// TIA Portal project "GME" (V18)

(* hardware
DEVICE "S7-1500/ET200MP station_1"  S7-1500 station
   slot 0: "Rail_0"  Rack  6ES7 590-1***0-0AA0
   slot 1: "102CPU"  CPU 1515-2 PN  6ES7 515-2AN03-0AB0  V3.0
      slot 3: "CPU display_1"  6ES7591-1BA00-0AA0
      slot 32768: "PROFINET interface_1"  X1
         slot 32769: "Port_1"  X1 P1
         slot 32770: "Port_2"  X1 P2
      slot 33024: "PROFINET interface_2"  X2
         slot 33025: "Port_1"  X2 P1
      slot 34817: "Virtual CP interface port_1"  Virtual CP interface port  Virtual CP interface port
   slot 2: "102A1"  AI 8xU/I/RTD/TC ST  6ES7 531-7KF00-0AB0  V2.2
   slot 3: "102A2"  AI 8xU/I/RTD/TC ST  6ES7 531-7KF00-0AB0  V2.2
   slot 4: "102A3"  AI 8xU/I/RTD/TC ST  6ES7 531-7KF00-0AB0  V2.2
   slot 5: "102A4"  AI 8xU/I/RTD/TC ST  6ES7 531-7KF00-0AB0  V2.2
   slot 6: "102A5"  AQ 8xU/I HS  6ES7 532-5HF00-0AB0  V2.2
   slot 7: "102A6"  AQ 8xU/I HS  6ES7 532-5HF00-0AB0  V2.2
   slot 8: "102A7"  DI 32x24VDC HF  6ES7 521-1BL00-0AB0  V2.2
   slot 9: "102A8"  DI 32x24VDC HF  6ES7 521-1BL00-0AB0  V2.2
   slot 10: "103A1"  DI 32x24VDC HF  6ES7 521-1BL00-0AB0  V2.2
   slot 11: "103A2"  DI 32x24VDC HF  6ES7 521-1BL00-0AB0  V2.2
   slot 12: "103A3"  DI 32x24VDC HF  6ES7 521-1BL00-0AB0  V2.2
   slot 13: "103GD1"  PS 25W 24VDC  6ES7 505-0KA00-0AB0  V1.0
   slot 14: "103A4"  DQ 32x24VDC/0.5A HF  6ES7 522-1BL01-0AB0  V1.1
   slot 15: "103A5"  DQ 32x24VDC/0.5A HF  6ES7 522-1BL01-0AB0  V1.1
   slot 16: "103A6"  TM Count 2x24V  6ES7 550-1AA01-0AB0  V2.0
   slot 17: "103A7"  TM Count 2x24V  6ES7 550-1AA01-0AB0  V2.0
   slot 18: "103A8"  TM Count 2x24V  6ES7 550-1AA01-0AB0  V2.0
DEVICE "S7-1500/ET200MP station_2"  S7-1500 station
   slot 0: "Rail_0"  Rack  6ES7 590-1***0-0AA0
   slot 1: "153IM155_JB1"  IM 155-5 PN ST  6ES7 155-5AA01-0AB0  V4.1
   slot 2: "153A1"  AI 8xU/I/RTD/TC ST  6ES7 531-7KF00-0AB0  V2.2
   slot 3: "153A2"  DQ 32x24VDC/0.5A HF  6ES7 522-1BL01-0AB0  V1.1
   slot 4: "153A3"  DI 16x24VDC/DQ 16x24VDC/0.5A BA  6ES7 523-1BL00-0AA0  V1.1
   slot 5: "153A4"  AQ 8xU/I HS  6ES7 532-5HF00-0AB0  V2.2
DEVICE "S7-1500/ET200MP station_3"  S7-1500 station
   slot 0: "Rail_0"  Rack  6ES7 590-1***0-0AA0
   slot 1: "182IM155_JB2"  IM 155-5 PN ST  6ES7 155-5AA01-0AB0  V4.1
   slot 2: "182A1"  DQ 32x24VDC/0.5A HF  6ES7 522-1BL01-0AB0  V1.1
   slot 3: "182A2"  DI 16x24VDC/DQ 16x24VDC/0.5A BA  6ES7 523-1BL00-0AA0  V1.1
*)

// ===== PLC "102CPU"  CPU 1515-2 PN =====

VAR_GLOBAL   // PLC tag table "Default tag table"
   "Main flame ON" AT %M25.0 : Bool;
   "Flag AutoBurner" AT %M15.0 : Bool;
   "Flag_Aggiorna_DB" AT %M1.7 : Bool;
   "Stop Counter PEW 336" AT %M114.3 : Bool;
   "Stop Counter PEW 368" AT %M115.3 : Bool;
   "Stop Counter PEW 418" AT %M116.3 : Bool;
   "TC01-TC02control disable" AT %M80.2 : Bool;
   "TC03 Close" AT %M40.7 : Bool;
   "TC03 Close2" AT %M41.1 : Bool;
   "TC03 Open" AT %M40.6 : Bool;
   "TC03 Open2" AT %M41.0 : Bool;
   "TEST CABIN" AT %M5.0 : Bool;
   "EV-82" AT %Q21.7 : Bool;   // A11.7 FILTER 8 VALVE BF02FOURTH SECTOR
   "EV-83" AT %Q22.0 : Bool;   // A12.0 FILTER 1 VALVE BF02FIFTH SECTOR
   "EV-84" AT %Q22.1 : Bool;   // A12.1 FILTER 2 VALVE BF02FIFTH SECTOR
   "EV-85" AT %Q22.2 : Bool;   // A12.2 FILTER 3 VALVE BF02FIFTH SECTOR
   "EV-87" AT %Q22.4 : Bool;   // A12.4 FILTER 5 VALVE BF02FIFTH SECTOR
   "EV-88" AT %Q22.5 : Bool;   // A12.5 FILTER 6 VALVE BF02FIFTH SECTOR
   "EV-89" AT %Q22.6 : Bool;   // A12.6 FILTER 7 VALVE BF02FIFTH SECTOR
   "EV-90" AT %Q22.7 : Bool;   // A12.7 FILTER 8 VALVE BF02FIFTH SECTOR
   "Module Access FLT" AT %M32.3 : Bool;
   "OB Fault" AT %M32.1 : Bool;
   "OFF" AT %M0.1 : Bool;
   "ON" AT %M0.0 : Bool;
   "OPEN MV05 PID" AT %M11.4 : Bool;
   "Every 1 second" AT %M1.0 : Bool;
   "Open EV A 00 PV-01" AT %M20.0 : Bool;
   "Open EV A 00 PV-02" AT %M30.4 : Bool;
   "Open EV A 01  PV-01" AT %M21.3 : Bool;
   "Riduce MN01" AT %M1.2 : Bool;
   "Scarico ceneri auto" AT %M15.1 : Bool;
   "Braking VS01" AT %Q49.5 : Bool;   // It's no longer there
   "Start Burner" AT %M48.3 : Bool;
   "PID DOWN MV04" AT %M14.3 : Bool;
   "PID DOWN MV05" AT %M13.1 : Bool;
   "PID MV02 Down" AT %M14.1 : Bool;
   "PID MV02 UP" AT %M14.0 : Bool;
   "PID UP MV03" AT %M14.4 : Bool;
   "PID UP MV04" AT %M14.2 : Bool;
   "PID UP MV05" AT %M13.0 : Bool;
   "PID down MV03" AT %M14.5 : Bool;
   "MEM2_0" AT %M2.0 : Bool;
   "MV WORK PULSE" AT %M10.0 : Bool;
   "WASHING MAX OK" AT %M9.0 : Bool;
   "PV-02 Gate ON" AT %M12.2 : Bool;
   "Close EV A 00  PV-01" AT %M20.2 : Bool;
   "Close EV A 01  PV-01" AT %M21.0 : Bool;
   "Close EV A 01  PV-02" AT %M30.0 : Bool;
   "Close EV A 02  PV-01" AT %M22.3 : Bool;
   "Close EV B 00  PV-01" AT %M20.3 : Bool;
   "Close EV B 01  PV-01" AT %M21.2 : Bool;
   "Close EV B 01  PV-02" AT %M30.2 : Bool;
   "Close EV B 02  PV-01" AT %M22.1 : Bool;
   "Close MV02 PID" AT %M11.7 : Bool;
   "Enable Counter PEW 336" AT %M114.2 : Bool;
   "Enable Counter PEW 368" AT %M115.2 : Bool;
   "Enable Counter PEW 418" AT %M116.2 : Bool;
   "Start VS01 BRAKE" AT %M11.0 : Bool;
   "Start client motor 4" AT %Q61.2 : Bool;   // It should be Free but it is used
   "Start client motor 6" AT %Q61.3 : Bool;   // It should be Free but it is used
   "Start client motor 8" AT %Q61.4 : Bool;   // It should be Free but it is used
   "Start client motor 9" AT %Q61.5 : Bool;   // It should be Free but it is used
   "Start client motore 10" AT %Q61.6 : Bool;   // It should be Free but it is used
   "EV-66" AT %Q19.7 : Bool;   // A9.7 FILTER 8 VALVE BF02SECOND SECTOR
   "EV-67" AT %Q20.0 : Bool;   // A10.0 FILTER 1 VALVE BF02THIRD SECTOR
   "EV-68" AT %Q20.1 : Bool;   // A10.1 FILTER 2 VALVE BF02THIRD SECTOR
   "EV-69" AT %Q20.2 : Bool;   // A10.2 FILTER 3 VALVE BF02THIRD SECTOR
   "EV-70" AT %Q20.3 : Bool;   // A10.3 FILTER 4 VALVE BF02THIRD SECTOR
   "EV-71" AT %Q20.4 : Bool;   // A10.4 FILTER 5 VALVE BF02THIRD SECTOR
   "EV-72" AT %Q20.5 : Bool;   // A10.5 FILTER 6 VALVE BF02THIRD SECTOR
   "EV-73" AT %Q20.6 : Bool;   // A10.6 FILTER 7 VALVE BF02THIRD SECTOR
   "EV-74" AT %Q20.7 : Bool;   // A10.7 FILTER 8 VALVE BF02THIRD SECTOR
   "EV-75" AT %Q21.0 : Bool;   // A11.0 FILTER 1 VALVE BF02FOURTH SECTOR
   "Open EV B 00  PV-02" AT %M30.5 : Bool;
   "Open EV B 01  PV-01" AT %M21.1 : Bool;
   "Open EV B 01  PV-02" AT %M30.1 : Bool;
   "Open EV B 02  PV-01" AT %M22.2 : Bool;
   "Open MV02 PID" AT %M11.6 : Bool;
   "PC01 Close" AT %M40.2 : Bool;
   "PC01 Open" AT %M40.3 : Bool;
   "PC02 Close" AT %M40.4 : Bool;
   "PC02 Open" AT %M40.5 : Bool;
   "m491" AT %M10.1 : Bool;
   "maintenance PV01" AT %M80.5 : Bool;
   "maintenance PV02" AT %M80.6 : Bool;
   "PLS M51 6" AT %M51.6 : Bool;
   "PLS M51.5" AT %M51.5 : Bool;
   "PLS M51_4" AT %M51.4 : Bool;
   "PLS m10.3" AT %M10.3 : Bool;
   "PLS m10.4" AT %M10.4 : Bool;
   "Button pushed" AT %M60.0 : Bool;
   "CLOSE MV05 PID" AT %M11.5 : Bool;
   "PLS 50 3" AT %M50.3 : Bool;
   "PLS 50 4" AT %M50.4 : Bool;
   "PLS 50 6" AT %M50.6 : Bool;
   "PLS 50 7" AT %M50.7 : Bool;
   "PLS 50_5" AT %M50.5 : Bool;
   "PLS 51 1" AT %M51.1 : Bool;
   "PLS 51 2" AT %M51.2 : Bool;
   "PLS 51 3" AT %M51.3 : Bool;
   "PLS M50.0" AT %M50.0 : Bool;
   "PLS M50.1" AT %M50.1 : Bool;
   "PLS M50.2" AT %M50.2 : Bool;
   "PLS M51 0" AT %M51.0 : Bool;
   "EV-76" AT %Q21.1 : Bool;   // A11.1 FILTER 2 VALVE BF02FOURTH SECTOR
   "EV-77" AT %Q21.2 : Bool;   // A11.2 FILTER 3 VALVE BF02FOURTH SECTOR
   "EV-78" AT %Q21.3 : Bool;   // A11.3 FILTER 4 VALVE BF02FOURTH SECTOR
   "EV-79" AT %Q21.4 : Bool;   // A11.4 FILTER 5 VALVE BF02FOURTH SECTOR
   "EV-80" AT %Q21.5 : Bool;   // A11.5 FILTER 6 VALVE BF02FOURTH SECTOR
   "EV-81" AT %Q21.6 : Bool;   // A11.6 FILTER 7 VALVE BF02FOURTH SECTOR
   "EV-51" AT %Q18.0 : Bool;   // A8.0 FILTER 1 VALVE BF02FIRST SECTOR
   "EV-52" AT %Q18.1 : Bool;   // A8.1 FILTER 2 VALVE BF02FIRST SECTOR
   "EV-53" AT %Q18.2 : Bool;   // A8.2 FILTER 3 VALVE BF02FIRST SECTOR
   "EV-54" AT %Q18.3 : Bool;   // A8.3 FILTER 4 VALVE BF02FIRST SECTOR
   "EV-55" AT %Q18.4 : Bool;   // A8.4 FILTER 5 VALVE BF02FIRST SECTOR
   "EV-56" AT %Q18.5 : Bool;   // A8.5 FILTER 6 VALVE BF02FIRST SECTOR
   "EV-57" AT %Q18.6 : Bool;   // A8.6 FILTER 7 VALVE BF02FIRST SECTOR
   "EV-58" AT %Q18.7 : Bool;   // A8.7 FILTER 8 VALVE BF02FIRST SECTOR
   "EV-59" AT %Q19.0 : Bool;   // A9.0 FILTER 1 VALVE BF02SECOND SECTOR
   "MV06 PID DOWN" AT %M13.3 : Bool;
   "MV06 PID UP" AT %M13.2 : Bool;
   "MEM Gate A OPEN PV-01" AT %M10.7 : Bool;
   "MEM Gate A OPEN PV-02" AT %M12.4 : Bool;
   "MEM Gate B OPEN PV-01" AT %M10.6 : Bool;
   "MEM Gate B OPEN PV-02" AT %M12.3 : Bool;
   "RO01 Close" AT %M40.1 : Bool;
   "RO01 Open" AT %M40.0 : Bool;
   "RO01-RO02control disable" AT %M80.1 : Bool;
   "RO01_CLOSE" AT %M41.3 : Bool;
   "RO01_OPEN" AT %M41.2 : Bool;
   "Rack FAULT" AT %M32.2 : Bool;
   "Reset Counter PEW 336" AT %M114.5 : Bool;
   "Reset Counter PEW 368" AT %M115.5 : Bool;
   "Reset Counter PEW 418" AT %M116.5 : Bool;
   "Disable masses" AT %M80.0 : Bool;
   "EV-61" AT %Q19.2 : Bool;   // A9.2 FILTER 3 VALVE BF02SECOND SECTOR
   "EV-86" AT %Q22.3 : Bool;   // A12.3 FILTER 4 VALVE BF02FIFTH SECTOR
   "I/O FLT" AT %M32.0 : Bool;
   "UNDER TESTING" AT %M5.5 : Bool;
   "Init_RK_512" AT %M200.0 : Bool;
   "UP MV01 PID" AT %M12.0 : Bool;
   "UP MV04 PID" AT %M11.2 : Bool;
   "APP M10.2" AT %M10.2 : Bool;
   "Enable start burner" AT %M48.2 : Bool;
   "Open MV03 for washing" AT %M48.1 : Bool;
   "Open false air" AT %M2.1 : Bool;
   "Programmed stop burner" AT %M1.1 : Bool;
   "Open EV A 01  PV-02" AT %M30.3 : Bool;
   "Open EV A 02  PV-01" AT %M22.0 : Bool;
   "Open EV B 00  PV-01" AT %M20.1 : Bool;
   "Enable start burner(1)" AT %M48.0 : Bool;
   "Prog FAULT" AT %M32.4 : Bool;
   "R1 Gate ON" AT %M10.5 : Bool;
   "Shot to close" AT %M18.0 : Bool;
   "Shot to open" AT %M18.1 : Bool;
   "Counter error PEW 336" AT %M114.4 : Bool;
   "Counter error PEW 368" AT %M115.4 : Bool;
   "Counter error PEW 418" AT %M116.4 : Bool;
   "DOWN MV01 PID" AT %M12.1 : Bool;
   "DOWN MV04 PID" AT %M11.3 : Bool;
   "DOWN TC03 PID MV04" AT %M11.1 : Bool;
   "Lock Burner" AT %M28.0 : Bool;
   "EV-60" AT %Q19.1 : Bool;   // A9.1 FILTER 2 VALVE BF02SECOND SECTOR
   "EV-62" AT %Q19.3 : Bool;   // A9.3 FILTER 4 VALVE BF02SECOND SECTOR
   "EV-63" AT %Q19.4 : Bool;   // A9.4 FILTER 5 VALVE BF02SECOND SECTOR
   "EV-64" AT %Q19.5 : Bool;   // A9.5 FILTER 6 VALVE BF02SECOND SECTOR
   "EV-65" AT %Q19.6 : Bool;   // A9.6 FILTER 7 VALVE BF02SECOND SECTOR
   "Tag_47" AT %T13 : Timer;
   "Tag_48" AT %T17 : Timer;
   "Tag_49" AT %T120 : Timer;
   "Tag_50" AT %T121 : Timer;
   "Tag_51" AT %T39 : Timer;
   "Tag_52" AT %T99 : Timer;
   "Tag_53" AT %T101 : Timer;
   "Tag_54" AT %T49 : Timer;
   "Tag_55" AT %T52 : Timer;
   "Tag_56" AT %T53 : Timer;
   "Tag_57" AT %T54 : Timer;
   "Tag_58" AT %T55 : Timer;
   "Tag_59" AT %T60 : Timer;
   "Tag_60" AT %T61 : Timer;
   "Tag_61" AT %T62 : Timer;
   "Tag_62" AT %T63 : Timer;
   "Tag_63" AT %T66 : Timer;
   "Tag_64" AT %T67 : Timer;
   "Tag_65" AT %T70 : Timer;
   "Tag_66" AT %T71 : Timer;
   "Tag_67" AT %T91 : Timer;
   "Tag_68" AT %T72 : Timer;
   "Tag_69" AT %T73 : Timer;
   "Tag_70" AT %T75 : Timer;
   "Tag_71" AT %T80 : Timer;
   "Tag_72" AT %T81 : Timer;
   "Tag_73" AT %T82 : Timer;
   "Tag_74" AT %T83 : Timer;
   "Tag_75" AT %T84 : Timer;
   "Tag_76" AT %T93 : Timer;
   "Tag_77" AT %T94 : Timer;
   "Tag_78" AT %T95 : Timer;
   "Tag_79" AT %T96 : Timer;
   "Tag_80" AT %T103 : Timer;
   "Tag_81" AT %T104 : Timer;
   "Tag_82" AT %T105 : Timer;
   "Tag_83" AT %T106 : Timer;
   "Tag_84" AT %T107 : Timer;
   "Tag_85" AT %T108 : Timer;
   "Tag_86" AT %T109 : Timer;
   "Tag_87" AT %T110 : Timer;
   "Tag_88" AT %T111 : Timer;
   "Tag_89" AT %T112 : Timer;
   "Tag_90" AT %T43 : Timer;
   "Tag_91" AT %T44 : Timer;
   "Tag_92" AT %T4 : Timer;
   "Tag_93" AT %T21 : Timer;
   "Tag_94" AT %T3 : Timer;
   "Tag_95" AT %T22 : Timer;
   "Tag_96" AT %T15 : Timer;
   "Tag_97" AT %T16 : Timer;
   "Tag_98" AT %T42 : Timer;
   "Tag_99" AT %T85 : Timer;
   "Tag_100" AT %T86 : Timer;
   "Tag_101" AT %T87 : Timer;
   "Tag_102" AT %T88 : Timer;
   "Tag_103" AT %T89 : Timer;
   "Tag_104" AT %T76 : Timer;
   "Tag_105" AT %T77 : Timer;
   "Tag_106" AT %T68 : Timer;
   "Tag_107" AT %T117 : Timer;
   "Tag_108" AT %T116 : Timer;
   "Tag_109" AT %T115 : Timer;
   "Tag_110" AT %T123 : Timer;
   "Tag_111" AT %T132 : Timer;
   "Tag_112" AT %T114 : Timer;
   "Tag_113" AT %T50 : Timer;
   "Tag_114" AT %T6 : Timer;
   "Tag_115" AT %T58 : Timer;
   "Tag_116" AT %T59 : Timer;
   "Tag_117" AT %T69 : Timer;
   "Tag_118" AT %T145 : Timer;
   "Tag_119" AT %T124 : Timer;
   "Tag_120" AT %T125 : Timer;
   "Tag_121" AT %T19 : Timer;
   "Tag_122" AT %T130 : Timer;
   "Tag_123" AT %T113 : Timer;
   "Tag_124" AT %T40 : Timer;
   "Tag_125" AT %T41 : Timer;
   "Tag_126" AT %T131 : Timer;
   "Tag_127" AT %T126 : Timer;
   "Tag_128" AT %T127 : Timer;
   "Tag_129" AT %T133 : Timer;
   "Tag_130" AT %T134 : Timer;
   "Tag_131" AT %T1 : Timer;
   "Tag_132" AT %T2 : Timer;
   "Tag_133" AT %T5 : Timer;
   "Tag_134" AT %T20 : Timer;
   "Tag_135" AT %T26 : Timer;
   "Tag_136" AT %T27 : Timer;
   "Tag_137" AT %T28 : Timer;
   "Tag_138" AT %T30 : Timer;
   "Tag_139" AT %T29 : Timer;
   "Tag_140" AT %T12 : Timer;
   "Tag_141" AT %T122 : Timer;
   "Tag_142" AT %T32 : Timer;
   "Tag_143" AT %T31 : Timer;
   "Tag_144" AT %T37 : Timer;
   "Tag_145" AT %T38 : Timer;
   "Tag_146" AT %T90 : Timer;
   "Tag_147" AT %T138 : Timer;
   "Tag_148" AT %T139 : Timer;
   "Tag_149" AT %T135 : Timer;
   "Tag_150" AT %T136 : Timer;
   "Tag_151" AT %T140 : Timer;
   "Tag_152" AT %T143 : Timer;
   "Tag_153" AT %T141 : Timer;
   "Tag_154" AT %T78 : Timer;
   "Tag_155" AT %T79 : Timer;
   "Tag_156" AT %T118 : Timer;
   "Tag_157" AT %T119 : Timer;
   "Tag_158" AT %MW70 : Word;
   "Tag_159" AT %T128 : Timer;
   "Tag_160" AT %T47 : Timer;
   "Tag_161" AT %T48 : Timer;
   "Tag_162" AT %T142 : Timer;
   "Tag_163" AT %T100 : Timer;
   "Tag_164" AT %T56 : Timer;
   "Tag_165" AT %T102 : Timer;
   "Tag_166" AT %T57 : Timer;
   "Tag_167" AT %T8 : Timer;
   "Tag_168" AT %T9 : Timer;
   "Tag_169" AT %T10 : Timer;
   "Tag_170" AT %T11 : Timer;
   "Tag_189" AT %MW80 : Word;
   "Tag_190" AT %MW82 : Word;
   "Tag_191" AT %M100.0 : Bool;
   "Tag_192" AT %M150.0 : Bool;
   "Tag_193" AT %M150.1 : Bool;
   "Tag_194" AT %M150.2 : Bool;
   "Tag_195" AT %M150.3 : Bool;
   "Tag_196" AT %M150.4 : Bool;
   "Tag_197" AT %M150.5 : Bool;
   "Tag_198" AT %M150.6 : Bool;
   "Tag_199" AT %M150.7 : Bool;
   "Tag_200" AT %M151.0 : Bool;
   "Tag_201" AT %M151.1 : Bool;
   "Tag_202" AT %M151.2 : Bool;
   "Tag_203" AT %M151.3 : Bool;
   "Tag_204" AT %M151.4 : Bool;
   "Tag_205" AT %M151.5 : Bool;
   "Tag_206" AT %M151.6 : Bool;
   "Tag_207" AT %M151.7 : Bool;
   "Tag_208" AT %M152.0 : Bool;
   "Tag_209" AT %M152.1 : Bool;
   "Tag_210" AT %M152.2 : Bool;
   "Tag_211" AT %M152.3 : Bool;
   "Tag_212" AT %M152.4 : Bool;
   "Tag_213" AT %M152.5 : Bool;
   "Tag_214" AT %M152.6 : Bool;
   "Tag_215" AT %M152.7 : Bool;
   "Tag_216" AT %M153.0 : Bool;
   "Tag_217" AT %M153.1 : Bool;
   "Tag_218" AT %M153.2 : Bool;
   "Tag_219" AT %M153.3 : Bool;
   "Tag_220" AT %M153.4 : Bool;
   "Tag_221" AT %M153.5 : Bool;
   "Tag_222" AT %M153.6 : Bool;
   "Tag_223" AT %M153.7 : Bool;
   "Tag_224" AT %M154.0 : Bool;
   "Tag_225" AT %M154.1 : Bool;
   "Tag_226" AT %M154.2 : Bool;
   "Tag_227" AT %M154.3 : Bool;
   "Tag_228" AT %M154.4 : Bool;
   "Tag_229" AT %M154.5 : Bool;
   "Tag_230" AT %M154.6 : Bool;
   "Tag_231" AT %M154.7 : Bool;
   "Tag_232" AT %M155.0 : Bool;
   "Tag_233" AT %M155.1 : Bool;
   "Tag_234" AT %M155.2 : Bool;
   "Tag_235" AT %M155.3 : Bool;
   "Tag_236" AT %M155.4 : Bool;
   "Tag_237" AT %M155.5 : Bool;
   "Tag_238" AT %M155.6 : Bool;
   "Tag_239" AT %M155.7 : Bool;
   "Tag_240" AT %M156.0 : Bool;
   "Tag_241" AT %M156.1 : Bool;
   "Tag_242" AT %M156.2 : Bool;
   "Tag_243" AT %M156.3 : Bool;
   "Tag_244" AT %M156.4 : Bool;
   "Tag_245" AT %M156.5 : Bool;
   "Tag_246" AT %M156.6 : Bool;
   "Tag_247" AT %M156.7 : Bool;
   "Tag_248" AT %M157.0 : Bool;
   "Tag_249" AT %M157.1 : Bool;
   "Tag_250" AT %M157.2 : Bool;
   "Tag_251" AT %M157.3 : Bool;
   "Tag_252" AT %M157.4 : Bool;
   "Tag_253" AT %M157.5 : Bool;
   "Tag_254" AT %M157.6 : Bool;
   "Tag_255" AT %M157.7 : Bool;
   "Tag_256" AT %M158.0 : Bool;
   "Tag_257" AT %M158.1 : Bool;
   "Tag_258" AT %M158.2 : Bool;
   "Tag_259" AT %M158.3 : Bool;
   "Tag_260" AT %M158.4 : Bool;
   "Tag_261" AT %M158.5 : Bool;
   "Tag_262" AT %M159.0 : Bool;
   "Tag_263" AT %M159.1 : Bool;
   "Tag_264" AT %M159.2 : Bool;
   "Tag_265" AT %M159.3 : Bool;
   "Tag_266" AT %M159.4 : Bool;
   "Tag_267" AT %M159.5 : Bool;
   "Tag_268" AT %M159.6 : Bool;
   "Tag_269" AT %M159.7 : Bool;
   "Tag_270" AT %M160.0 : Bool;
   "Tag_271" AT %M160.1 : Bool;
   "Tag_272" AT %M160.2 : Bool;
   "Tag_273" AT %M160.3 : Bool;
   "Tag_280" AT %QW0 : Word;
   "Tag_281" AT %QW2 : Word;
   "Tag_282" AT %QW4 : Word;
   "Tag_283" AT %QW6 : Word;
   "Tag_284" AT %QW8 : Word;
   "Tag_285" AT %QW10 : Word;
   "Tag_286" AT %QW12 : Word;
   "Tag_287" AT %QW14 : Word;
   "Tag_288" AT %QW16 : Word;
   "Tag_289" AT %QW18 : Word;
   "Tag_290" AT %QW20 : Word;
   "Tag_291" AT %QW22 : Word;
   "Simulation(1)" AT %M180.0 : Bool;
   "Clock100ms" AT %M90.0 : Bool;
   "Clock3s" AT %M90.1 : Bool;
   "Tag_292" AT %M90.5 : Bool;
   "ServiceBit" AT %M1000.0 : Bool;   // must be always false
   "Clock_Byte" AT %MB2000 : Byte;
   "Clock_10Hz" AT %M2000.0 : Bool;
   "Clock_5Hz" AT %M2000.1 : Bool;
   "Clock_2.5Hz" AT %M2000.2 : Bool;
   "Clock_2Hz" AT %M2000.3 : Bool;
   "Clock_1.25Hz" AT %M2000.4 : Bool;
   "Clock_1Hz" AT %M2000.5 : Bool;
   "Clock_0.625Hz" AT %M2000.6 : Bool;
   "Clock_0.5Hz" AT %M2000.7 : Bool;
   "Memo_M25_Running" AT %M180.1 : Bool;
   "FP_M25_Run" AT %M180.2 : Bool;
   "BF01_RUN" AT %M180.3 : Bool;
   "BF02_RUN" AT %M180.4 : Bool;
   "Close MV03 for Burner Startup" AT %M180.5 : Bool;
   "MemoCMD_PV1_Startup" AT %M180.6 : Bool;
   "MemoCMD_BC01_Startup" AT %M180.7 : Bool;
   "PS181_0" AT %M181.0 : Bool;
END_VAR

VAR_GLOBAL   // PLC tag table "Input"
   "TC04" AT %IW256 : Int;
   "RESERVED TC04" AT %IW258 : Int;
   "TC05" AT %IW260 : Int;   // PROBE SENSOR PT100 BEARING FN-01 (TC-04) -30...250°C
   "RESERVED TC05" AT %IW262 : Int;   // PROBE SENSOR PT100 BEARING FN-01 (TC-05) -30...350°C
   "BWF01_FlowRate" AT %IW264 : Int;   // FLOW RATE BWF 01(CLIENT MACHINE)
   "BWF02_FlowRate" AT %IW266 : Int;   // FLOW RATE BWF 02 (CLIENT MACHINE)
   "BWF01_Level" AT %IW268 : Int;   // LEVEL BWF 01 (CLIENT MACHINE)
   "BWF02_Level" AT %IW270 : Int;   // LEVEL BWF 02 (CLIENT MACHINE)
   "TC01" AT %IW272 : Int;   // TEMPERATURE CHAMBER AB-01
   "TC02" AT %IW274 : Int;   // SAFETY TEMPERATURE CHAMBER AB-01
   "TC03" AT %IW276 : Int;   // TEMPERATURE CONTROL OUTPUTSMOKE
   "TC06" AT %IW278 : Int;   // TEMPERATURE CONTROL OUTPUTAB-01
   "TC07" AT %IW280 : Int;   // TEMPERATURE CONTROL INPUTSMOKE
   "ZT01" AT %IW282 : Int;   // VIBRATION TRASMITTER BLOWER FN-01
   "PSH01" AT %IW284 : Int;   // PRESSURE CONTROL OUTPUT MV-02
   "PSH02" AT %IW286 : Int;   // PRESSURE CONTROL OUTPUT MV-03
   "PSH03" AT %IW320 : Int;   // PRESSURE CONTROL
   "PC01" AT %IW322 : Int;   // PRESSURE CONTROL
   "MV04_M18A" AT %IW324 : Int;   // MV-04 POSITION M18A
   "MV04_M18B" AT %IW326 : Int;   // MV-04 POSITION M18B
   "FN02_Current" AT %IW328 : Int;   // BLOWER FAN CURRENT
   "102A3_SPARE0" AT %IW330 : Int;
   "RD01_Current" AT %IW332 : Int;   // ROTATING DRUM CURRENT
   "FN01_Current" AT %IW334 : Int;   // BLOWER FAN CURRENT FN-01
   "R001" AT %IW352 : Int;   // OXIGEN CONTROL
   "R002" AT %IW354 : Int;   // OXIGEN CONTROL
   "R003" AT %IW356 : Int;   // OXIGEN CONTROL
   "R004" AT %IW358 : Int;   // OXIGEN CONTROL
   "BR01_GAS" AT %IW360 : Int;   // GAS SERVO-MOTOR BR-01
   "BR01_AIR" AT %IW362 : Int;   // AIR SERVO-MOTOR BR-01
   "BR01_FlowMeter_GAS" AT %IW364 : Int;   // GAS OUTLET BR-01
   "BR01_FlowMeter_AIR" AT %IW366 : Int;   // AIR OUTLET BR-01
   "BC01_Fbk" AT %I0.0 : Bool;   // FEEDBACK MOTOR BC-01
   "BC01_All_inv" AT %I0.1 : Bool;   // ALARM MOTOR BC-01
   "RD01_Fbk" AT %I0.2 : Bool;   // FEEDBACK MOTOR RD-01
   "RD01_All_inv" AT %I0.3 : Bool;   // ALARM MOTOR RD-01
   "RD01F_Fbk" AT %I0.4 : Bool;   // FEEDBACK MOTOR RD-01F
   "102A7_SPARE5" AT %I0.5 : Bool;
   "MC04_Fbk" AT %I0.6 : Bool;   // FEEDBACK MOTOR MC-04
   "MC04_All_inv" AT %I0.7 : Bool;   // FEEDBACK MOTOR MC-04
   "MC05_Fbk" AT %I1.0 : Bool;   // FEEDBACK MOTOR MC-05
   "VS01_Fbk" AT %I1.1 : Bool;   // FEEDBACK MOTOR VS-01/VS-01A
   "VS01_All_Inv" AT %I1.2 : Bool;   // ALARM MOTOR VS-01/VS-01A
   "SC12_Fbk" AT %I1.3 : Bool;   // FEEDBACK MOTOR SC-12
   "MV02_05_06_POWER_OK" AT %I1.4 : Bool;   // FEEDBACK INVERTER SUPPLY MOTORS MV-02/MV-05/MV-06
   "MV02_05_06_Inv_All" AT %I1.5 : Bool;   // ALARM INVERTER SUPPLY MOTORS MV-02/MV-05/MV-06
   "MV06_Fbk_Opening" AT %I1.6 : Bool;   // FEEDBACK OPENING MOTOR MV-06
   "MV06_Fbk_Closing" AT %I1.7 : Bool;   // FEEDBACK CLOSING MOTOR MV-06
   "MV05_Fbk_Opening" AT %I2.0 : Bool;   // FEEDBACK OPENING MOTOR MV-05
   "MV05_Fbk_Closing" AT %I2.1 : Bool;   // FEEDBACK CLOSING MOTOR MV-05
   "MV02_Fbk_Opening" AT %I2.2 : Bool;   // FEEDBACK OPENING MOTOR MV-02
   "MV02_Fbk_Closing" AT %I2.3 : Bool;   // FEEDBACK CLOSING MOTOR MV-02
   "MV03_Fbk_Opening" AT %I2.4 : Bool;   // FEEDBACK OPENING MOTOR MV-03
   "MV03_Fbk_Closing" AT %I2.5 : Bool;   // FEEDBACK CLOSING MOTOR MV-03
   "MV04_Fbk_Opening" AT %I2.6 : Bool;   // FEEDBACK OPENING MOTOR MV-04
   "MV04_Fbk_Closing" AT %I2.7 : Bool;   // FEEDBACK CLOSING MOTOR MV-04
   "FN02_Fbk" AT %I3.0 : Bool;   // FEEDBACK MOTOR FN-02
   "FN02_All_Inv" AT %I3.1 : Bool;   // ALARM MOTOR FN-02
   "MV01_Fbk_Opening" AT %I3.2 : Bool;   // FEEDBACK OPENINGMOTOR MV-01
   "MV01_Fbk_Closing" AT %I3.3 : Bool;   // FEEDBACK CLOSINGMOTOR MV-01
   "VR01_Fbk" AT %I3.4 : Bool;   // FEEDBACKMOTOR VR-01
   "FN01_Fbk" AT %I3.5 : Bool;   // FEEDBACKMOTOR FN-01
   "FN01_All_Inv" AT %I3.6 : Bool;   // ALARM MOTOR FN-01
   "VR02_Fbk" AT %I3.7 : Bool;   // FEEDBACKMOTOR VR-02
   "CH01_Fbk" AT %I4.0 : Bool;   // FEEDBACK MOTOR CH-01
   "FN03_Fbk" AT %I4.1 : Bool;   // FEEDBACK MOTOR FN-03
   "FN03_All_SoftStarter" AT %I4.2 : Bool;   // ALARM MOTOR FN-03
   "FN06_Fbk" AT %I4.3 : Bool;   // FEEDBACK MOTOR FN-06
   "SC01_Fbk" AT %I4.4 : Bool;   // FEEDBACK MOTOR SC-01
   "FN01F_Fbk" AT %I4.5 : Bool;   // FEEDBACK COOLING FAN MOTOR FN-01
   "LD-01_Fbk" AT %I4.6 : Bool;   // FEEDBACK MOTOR LD-01
   "LD-01A_Fbk" AT %I4.7 : Bool;   // FEEDBACK MOTOR-LD-01A
   "SC-10_Fbk" AT %I5.0 : Bool;   // FEEDBACK MOTOR SC-10
   "SC-11_Fbk" AT %I5.1 : Bool;   // FEEDBACK MOTOR SC-11
   "102A8_SPARE0" AT %I5.2 : Bool;
   "102A8_SPARE1" AT %I5.3 : Bool;
   "VR03_Fbk" AT %I5.4 : Bool;   // FEEDBACK MOTOR VR-03
   "VR04_Fbk" AT %I5.5 : Bool;   // FEEDBACK MOTOR VR-04
   "VR05_Fbk" AT %I5.6 : Bool;   // FEEDBACK MOTOR VR-05
   "VR06_Fbk" AT %I5.7 : Bool;   // FEEDBACK MOTOR VR-06
   "FN05_Fbk" AT %I6.0 : Bool;   // FEEDBACK MOTOR FN-05
   "ER01_Fbk" AT %I6.1 : Bool;   // FEEDBACK ER-01 ELECTRICAL RESISTANCE
   "BC01_TripWire" AT %I6.2 : Bool;   // LIMIT SWITCH SS-01
   "BC01_Prox" AT %I6.3 : Bool;   // LIMIT SWITCH SSL-01
   "MC03_torque" AT %I6.4 : Bool;   // LIMIT SWITCH SS-09
   "MC04_torque" AT %I6.5 : Bool;   // LIMIT SWITCH SS-10
   "MC05_torque" AT %I6.6 : Bool;   // LIMIT SWITCH SS-11
   "MV06_Open" AT %I6.7 : Bool;   // LIMIT SWITCH LS.40
   "MV06_Close" AT %I7.0 : Bool;   // LIMIT SWITCH LS-41
   "MV05_Open" AT %I7.1 : Bool;   // LIMIT SWITCH LS-15
   "MV05_Close" AT %I7.2 : Bool;   // LIMIT SWITCH LS-16
   "MV02_Open" AT %I7.3 : Bool;   // LIMIT SWITCH LS-17
   "MV02_Close" AT %I7.4 : Bool;   // LIMIT SWITCH LS-18
   "MV03_Open" AT %I7.5 : Bool;   // LIMIT SWITCH LS-19
   "MV03_Close" AT %I7.6 : Bool;   // LIMIT SWITCH LS-20
   "MV04_Open" AT %I7.7 : Bool;   // LIMIT SWITCH LS21A/LS21B
   "MV04_Close" AT %I8.0 : Bool;   // LIMIT SWITCH LS-22A/LS-22B
   "MV01_Open" AT %I8.1 : Bool;   // LIMIT SWITCH LS-23
   "MV01_Close" AT %I8.2 : Bool;   // LIMIT SWITCH LS-24
   "102A9_SPARE0" AT %I8.3 : Bool;
   "102A9_SPARE1" AT %I8.4 : Bool;
   "102A9_SPARE2" AT %I8.5 : Bool;
   "EV01_Open" AT %I8.6 : Bool;   // LIMIT SWITCH LS-01 GATE "A" OPEN
   "EV01_Close" AT %I8.7 : Bool;   // LIMIT SWITCH LS-02 GATE "A" CLOSED
   "EV02_Open" AT %I9.0 : Bool;   // LIMIT SWITCH LS-05 GATE "B" OPEN
   "EV02_Close" AT %I9.1 : Bool;   // LIMIT SWITCH LS-06 GATE "B" CLOSED
   "EV01_Sel_Open" AT %I9.2 : Bool;   // OPENING GATE "A"LOCAL SELECTOR
   "EV02_Sel_Open" AT %I9.3 : Bool;   // OPENING GATE "B"LOCAL SELECTOR
   "EV04_Open" AT %I9.4 : Bool;   // E29.6 LIMIT SWITCH LS-25GATE "A" OPEN
   "EV04_Close" AT %I9.5 : Bool;   // E29.7 LIMIT SWITCH LS-26GATE "A" CLOSED
   "EV05_Open" AT %I9.6 : Bool;   // E29.2 LIMIT SWITCH LS-29GATE "B" OPEN
   "EV05_Close" AT %I9.7 : Bool;   // E29.3 LIMIT SWITCH LS-30GATE "B" CLOSED
   "Selector Op Gate A PV-02" AT %I10.0 : Bool;   // E45.4 OPENING GATE "A"LOCAL SELECTOR
   "Selector Op Gate B PV-02" AT %I10.1 : Bool;   // E45.5 OPENING GATE "B"LOCAL SELECTOR
   "Deviator Open PV-03" AT %I10.2 : Bool;   // E29.4 LIMIT SWITCHLS-09
   "Deviator Close PV-03" AT %I10.3 : Bool;   // E29.5 LIMIT SWITCHLS-10
   "PV03 Local Selector" AT %I10.4 : Bool;   // E65.7 73SA1 DEVIATOREV-06 SELECTOR
   "PV04 Open" AT %I10.5 : Bool;   // E 45.0 pv 04 ls33 open
   "PV04 Close" AT %I10.6 : Bool;   // E36.6 LIMIT SWITCHLS-32
   "Button Open PV-0000" AT %I10.7 : Bool;   // E 37.6 74SB1 diverterV-07 SELECTOR
   "Low Pressure Air" AT %I11.0 : Bool;   // E 41.4 PSL-05 LOW AIRPRESSURE SWITCH
   "BWF01 OK" AT %I11.1 : Bool;   // E 64.0 BWF 01 MANU STATUS
   "BWF 01 RUN" AT %I11.2 : Bool;   // E 64.1 BWF 01 RUN
   "BWF01 FAULT" AT %I11.3 : Bool;   // E 64.2 BWF 01 FAULT
   "min LEV BWF01" AT %I11.4 : Bool;   // E 64.3 BWF 01 MINIMUM LEVEL
   "MAX LEV BWF01" AT %I11.5 : Bool;   // E 64.4 BWF 01MAXIMUM LEVEL
   "BWF02 OK" AT %I11.6 : Bool;   // E 64.5 BWF 02 MANU STATUS
   "BWF 02 RUN" AT %I11.7 : Bool;   // E 64.6 BWF 02 RUN
   "BWF02 FAULT" AT %I12.0 : Bool;   // E 64.7 BWF 02 FAULT
   "min LEV BWF02" AT %I12.1 : Bool;   // E 65.0 BWF 02MINIMUM LEVEL
   "MAX LEV BWF02" AT %I12.2 : Bool;   // E 65.1 BWF 02MAXIMUM LEVEL
   "APRON CONVEYOR A RUN" AT %I12.3 : Bool;   // E 13.0 APRON CONVEYOR "A"RUN
   "IMPACTOR RUN" AT %I12.4 : Bool;   // E 13.1 IMPACTOR RUN
   "IMPACT VIBRATIONFEEDER RUN" AT %I12.5 : Bool;   // E 13.2 IMPACT VIBRATIONFEEDER RUN
   "BELT CONVEYOR A RUN" AT %I12.6 : Bool;   // E 13.3 BELT CONVEYOR "A"RUN
   "AIR KNIFE RUN" AT %I12.7 : Bool;   // E 13.4 AIR KNIFE RUN
   "BELT CONVEYOR B RUN" AT %I13.0 : Bool;   // E 13.5 BELT CONVEYOR "B"RUN
   "SHREDDER 1 RUN" AT %I13.1 : Bool;   // E 13.6 SHREDDER 1 RUN
   "SHREDDER VIBRATIONFEEDER RUN" AT %I13.2 : Bool;   // E 13.7 SHREDDER VIBRATIONFEEDER RUN
   "BELT CONVEYOR  C RUN" AT %I13.3 : Bool;   // E 14.0 BELT CONVEYOR "C"RUN
   "ROTEX SCREEN RUN" AT %I13.4 : Bool;   // E 14.1 ROTEX SCREEN RUN
   "APRON CONVEYOR B RUN" AT %I13.5 : Bool;   // E 14.4 APRON CONVEYOR "B"RUN
   "SHREDDER 2 RUN" AT %I13.6 : Bool;   // E 14.5 SHREDDER 2 RUN
   "BELT CONVEYOR  D RUN" AT %I13.7 : Bool;   // E 14.6 BELT CONVEYOR "D"RUN
   "BELT CONVEYOR E RUN" AT %I14.0 : Bool;   // E 14.7 BELT CONVEYOR "E"RUN
   "LIW SYSTEMAUTOREADER" AT %I14.1 : Bool;   // E 15.0 LIW SYSTEMAUTOREADER
   "PRIMARYSHREDDER RUN" AT %I14.2 : Bool;   // E 15.2 PRIMARYSHREDDER RUN
   "102A10_SPARE0" AT %I14.3 : Bool;   // CONSENT SPARE
   "BWF1_INVERTER_HIGH_SPEED" AT %I14.4 : Bool;   // E 17.0 BWF1_INVERTER_HIGH_SPEED
   "BWF2_INVERTER_HIGH_SPEED" AT %I14.5 : Bool;   // E 17.1 BWF2_INVERTER_HIGH_SPEED
   "APRON CONVEYOR A FAULT" AT %I14.6 : Bool;   // E 17.6 APRON CONVEYOR "A"FAULT
   "IMPACTOR FAULT" AT %I14.7 : Bool;   // E 17.7 IMPACTOR FAULT
   "IMPACT VIBRATIONFEEDER FAULT" AT %I15.0 : Bool;   // E 18.0 IMPACT VIBRATIONFEEDER FAULT
   "BELT CONVEYOR  A FAULT" AT %I15.1 : Bool;   // E 18.1 BELT CONVEYOR "A"FAULT
   "AIR KNIFE FAULT" AT %I15.2 : Bool;   // E 18.2 AIR KNIFE FAULT
   "BELT CONVEYOR B FAULT" AT %I15.3 : Bool;   // E 18.3 BELT CONVEYOR "B"FAULT
   "SHREDDER 1 FAULT" AT %I15.4 : Bool;   // E 18.4 SHREDDER 1 FAULT
   "SHREDDER VIBRATIONFEEDER FAULT" AT %I15.5 : Bool;   // E 18.5 SHREDDER VIBRATIONFEEDER FAULT
   "BELT CONVEYOR C FAULT" AT %I15.6 : Bool;   // E 18.6 BELT CONVEYOR "C"FAULT
   "ROTEX SCREENFAULT" AT %I15.7 : Bool;   // E 18.7 ROTEX SCREENFAULT
   "APRON CONVEYOR B FAULT" AT %I16.0 : Bool;   // E19.2 APRON CONVEYOR "B"FAULT
   "SHREDDER 2FAULT" AT %I16.1 : Bool;   // E19.3 SHREDDER 2FAULT
   "BELT COVEYOR  D FAULT" AT %I16.2 : Bool;   // E19.4 BELT COVEYOR "D"FAULT
   "BELT CONVEYOR  E FAULT" AT %I16.3 : Bool;   // E19.5 BELT CONVEYOR "E"FAULT
   "WEIGHTING HOPPER 2FAULT" AT %I16.4 : Bool;   // E19.6 WEIGHTING HOPPER 2FAULT
   "HOPPER CONVEYOR 2FAULT" AT %I16.5 : Bool;   // E19.7 HOPPER CONVEYOR 2FAULT
   "BELT CONVEYOR C FAULT_doppio!" AT %I16.6 : Bool;   // E20.0 BELT CONVEYOR "C"FAULT
   "NITROGEN TANK READY" AT %I16.7 : Bool;   // E 45.7 NITROGEN TANKREADY
   "Burner On" AT %I17.0 : Bool;   // E 44.7 BURNER ON
   "Brurner Lock Out" AT %I17.1 : Bool;   // E 44.6 BURNER LOCKOUT
   "Burner ON and OK" AT %I17.2 : Bool;   // E 44.1 BURNER INMODULATION
   "Min Pressure Gas" AT %I17.3 : Bool;   // E 44.2 LIMIT SWITCH S3MIN.PRESSURE GAS
   "Max Pressure Gas" AT %I17.4 : Bool;   // E 44.3 LIMIT SWITCH S4MAX PRESSURE GAS
   "Min Pressure Air" AT %I17.5 : Bool;   // E 44.4 LIMIT SWITCH S3MIN.PRESSURE AIR
   "Max Pressure Air" AT %I17.6 : Bool;   // E 40.6 LIMIT SWITCH S4MAX PRESSURE AIR
   "High Flame Gas" AT %I17.7 : Bool;   // E 41.7 HIGH FLAME GASVALVE INSERTED
   "103A3_SPARE0" AT %I18.0 : Bool;
   "103A3_SPARE1" AT %I18.1 : Bool;
   "103A3_SPARE2" AT %I18.2 : Bool;
   "103A3_SPARE3" AT %I18.3 : Bool;
   "103A3_SPARE4" AT %I18.4 : Bool;
   "103A3_SPARE5" AT %I18.5 : Bool;
   "103A3_SPARE6" AT %I18.6 : Bool;
   "103A3_SPARE7" AT %I18.7 : Bool;
   "103A3_SPARE8" AT %I19.0 : Bool;
   "103A3_SPARE9" AT %I19.1 : Bool;
   "103A3_SPARE10" AT %I19.2 : Bool;
   "103A3_SPARE11" AT %I19.3 : Bool;
   "EM_OK" AT %E19.4 : Bool;
   "Presence 110V" AT %E19.5 : Bool;
   "acknowledg" AT %I19.6 : Bool;
   "Reset_allarm" AT %I19.7 : Bool;
   "TC09" AT %IW386 : Int;   // TEMPERATURE BF-01
   "TC-10" AT %IW390 : Int;   // SPARE TEMPERATURE
   "153A1_SPARE1" AT %IW392 : Int;
   "FN04_Current" AT %IW394 : Int;   // MAIN ASPIRATOR ABSORPTION CURRENT FN-04(4-20mA)
   "153A1_SPARE3" AT %IW396 : Int;
   "PR_BF01" AT %IW398 : Int;   // DIFFERENTIAL PRESSURE SWITCHBAGS FILTER BF-01(4-20mA)
   "PR_BR02" AT %IW400 : Int;   // DIFFERENTIAL PRESSURE SWITCHBAGS FILTER BF-02(4-20mA)
   "PV-14 OPEN" AT %I28.0 : Bool;   // %I6.0
   "PV-14 CLOSE" AT %I28.1 : Bool;   // %I6.1
   "FN04_Fbk" AT %I28.2 : Bool;
   "FN04_All_inv" AT %I28.3 : Bool;
   "177T1_OK" AT %I28.4 : Bool;
   "LL_LD01" AT %I28.5 : Bool;
   "170FC1" AT %I28.6 : Bool;
   "170SA1" AT %I28.7 : Bool;
   "153A3_SPARE0" AT %I29.0 : Bool;
   "153A3_SPARE1" AT %I29.1 : Bool;
   "153A3_SPARE2" AT %I29.2 : Bool;
   "153A3_SPARE3" AT %I29.3 : Bool;
   "153A3_SPARE4" AT %I29.4 : Bool;
   "153A3_SPARE5" AT %I29.5 : Bool;
   "153A3_SPARE6" AT %I29.6 : Bool;
   "153A3_SPARE7" AT %I29.7 : Bool;
   "Tag_178" AT %IW0 : Word;
   "Tag_179" AT %IW2 : Word;
   "Tag_180" AT %IW4 : Word;
   "Tag_171" AT %IW6 : Word;
   "Tag_181" AT %IW8 : Word;
   "Tag_182" AT %IW10 : Word;
   "Tag_183" AT %IW12 : Word;
   "Tag_274" AT %IW14 : Word;
   "Tag_275" AT %IW16 : Word;
   "Tag_276" AT %IW18 : Word;
   "Tag_277" AT %IW20 : Word;
   "BWF01 Pulse" AT %I20.1 : Bool;   // Old address
   "BWF02 Pulse" AT %I20.2 : Bool;   // Old address
   "Tag_278" AT %IW22 : Word;
   "Tag_279" AT %IW24 : Word;
   "Tag_172" AT %IW28 : Word;
   "Tag_173" AT %IW32 : Word;
   "Tag_174" AT %IW36 : Word;
   "Free E37.0" AT %I37.0 : Bool;
   "Tag_175" AT %IW40 : Word;
   "Tag_176" AT %IW44 : Word;
   "Free E45.1" AT %I45.1 : Bool;
   "Tag_184" AT %IW48 : Word;
   "Tag_185" AT %IW52 : Word;
   "Tag_186" AT %IW56 : Word;
   "Tag_187" AT %IW60 : Word;
   "Tag_177" AT %IW64 : Word;
   "Tag_188" AT %IW68 : Word;
END_VAR

VAR_GLOBAL   // PLC tag table "Output"
   "Start BC01" AT %Q0.0 : Bool;   // A 48.1 BC-01 MOTORCOMMAND
   "Start RD01" AT %Q0.1 : Bool;   // A 48.5 RD-01 MOTORCOMMAND
   "Start fan RD01" AT %Q0.2 : Bool;   // A 48.6 RD-01F MOTORCOMMAND
   "Start Spare Motor" AT %Q0.3 : Bool;   // A 48.7 SPARE MOTORCOMMAND
   "Start MC04" AT %Q0.4 : Bool;   // A 49.1 MC-04 MOTORCOMMAND
   "Start MC05" AT %Q0.5 : Bool;   // A 49.2 MC-05 MOTORCOMMAND
   "Start VS01" AT %Q0.6 : Bool;   // A 49.0 VS-01/VS-01AMOTOR COMMAND
   "Start SC12" AT %Q0.7 : Bool;   // A 48.0 SC-12 MOTORCOMMAND
   "Start Aux INV" AT %Q1.0 : Bool;   // Start Inverter for Valve Motorized MV02-05-06
   "Open MV06" AT %Q1.1 : Bool;   // A 60.6 MV-06 OPENINGMOTOR COMMAND
   "Close MV06" AT %Q1.2 : Bool;   // A 60.7 MV-06 CLOSINGMOTOR COMMAND
   "Open MV05" AT %Q1.3 : Bool;   // A 48.2 MV-05 OPENINGMOTOR COMMAND
   "Close MV05" AT %Q1.4 : Bool;   // A 48.3 MV-05 CLOSINGMOTOR COMMAND
   "Open MV02" AT %Q1.5 : Bool;   // A 57.2 MV-02 OPENINGMOTOR COMMAND
   "Close MV02" AT %Q1.6 : Bool;   // A 57.3 MV-02 CLOSINGMOTOR COMMAND
   "Start open MV03" AT %Q1.7 : Bool;   // A 52.5 MV-03 OPENINGMOTOR COMMAND
   "Start Close MV03" AT %Q2.0 : Bool;   // A 52.6 MV-03 CLOSINGMOTOR COMMAND
   "Open MV04" AT %Q2.1 : Bool;   // A 57.4 MV-04 OPENINGMOTOR COMMAND
   "Close MV04" AT %Q2.2 : Bool;   // A 57.5 MV-04 CLOSINGMOTOR COMMAND
   "Start FN02" AT %Q2.3 : Bool;   // A 52.0 FN-02 MOTORCOMMAND
   "Start Open MV-01" AT %Q2.4 : Bool;   // A 60.1 MV-01 OPENINGMOTOR COMMAND
   "Start Close MV-01" AT %Q2.5 : Bool;   // A 60.2 MV-01 CLOSINGMOTOR COMMAND
   "Start VR01" AT %Q2.6 : Bool;   // A 53.2 VR-01 MOTORCOMMAND
   "Start FN01" AT %Q2.7 : Bool;   // A 49.6 FN-01 MOTORCOMMAND
   "Start VR02" AT %Q3.0 : Bool;   // A 49.7 VR-02 MOTORCOMMAND
   "Start CH01" AT %Q3.1 : Bool;   // A 53.4 CH-01 MOTORCOMMAND
   "Start FN03" AT %Q3.2 : Bool;   // A 56.0 FN-03 MOTORCOMMAND
   "Start FN06" AT %Q3.3 : Bool;   // A 60.3 FN-06 MOTORCOMMAND
   "Start SC01" AT %Q3.4 : Bool;   // A 49.3 SC-01 MOTORCOMMAND
   "Star fan FN01" AT %Q3.5 : Bool;   // A 53.5 FN-01 MOTORCOMMAND cooling fan
   "Start LD01" AT %Q3.6 : Bool;   // A 49.4 LD-01 MOTORCOMMAND
   "Start Vibrator LD-01" AT %Q3.7 : Bool;   // A 52.1 LD-01A MOTORCOMMAND
   "Start SC10" AT %Q4.0 : Bool;   // A 52.2 SC-10 MOTORCOMMAND
   "Start SC11" AT %Q4.1 : Bool;   // A 52.3 SC-11 MOTORCOMMAND
   "Spare_0" AT %Q4.2 : Bool;   // A 52.4 FN-04/FN-04A MOTORCOMMAND
   "Start VR03" AT %Q4.3 : Bool;   // A 52.7 VR-03 MOTORCOMMAND
   "Start VR04" AT %Q4.4 : Bool;   // A 53.0 VR-04 MOTORCOMMAND
   "Start VR05" AT %Q4.5 : Bool;   // A 53.3 VR-05 MOTORCOMMAND
   "Start VR06" AT %Q4.6 : Bool;   // A 53.6 VR-06 MOTORCOMMAND
   "Start FN05" AT %Q4.7 : Bool;   // A 60.0 FN-05 MOTORCOMMAND
   "Start ER-01" AT %Q5.0 : Bool;   // A 60.4 ER-01 ELECTRICALRESISTANCE COMMAND
   "EV03" AT %Q5.1 : Bool;   // A 53.1 EV-03 VALVECOMMAND
   "PV-01 Gate a" AT %Q5.2 : Bool;   // A 57.0 EV-01 VALVECOMMAND
   "PV-01 GATE B EV" AT %Q5.3 : Bool;   // A 48.4 EV-02 VALVECOMMAND
   "PV-02 GATE A EV" AT %Q5.4 : Bool;   // A 53.7 EV-04 VALVECOMMAND
   "PV-02 GATE B EV" AT %Q5.5 : Bool;   // A 56.4 EV-05 VALVECOMMAND
   "PV-03 GATE EV" AT %Q5.6 : Bool;   // A 56.5 EV-06 VALVECOMMAND
   "PV-04" AT %Q5.7 : Bool;   // A 57.1 EV-07 VALVECOMMAND
   "Enable start chiller" AT %Q6.0 : Bool;   // A 61.0 CHILLER REMOTESTART
   "START LIW FEEDER" AT %Q6.1 : Bool;   // A 61.1 LIW FEEDERREMOTE START
   "Consent Start BWF01" AT %Q6.2 : Bool;   // A 61.7 BWF 01 REMOTESTART
   "Consent Start BWF02" AT %Q6.3 : Bool;   // A 68.3 BWF 02 REMOTESTART
   "Start Nitrogen" AT %Q6.4 : Bool;   // A 60.5 AUTOMATIC IMMISSIONMOTOR COMMAND
   "Rem. Start/Stop Burner" AT %Q6.5 : Bool;   // A 56.1 REMOTE START/STOPBURNER
   "Temperature Interlock OK" AT %Q6.6 : Bool;   // A 56.3 MAX.TEMPERATUREFILTER
   "Rst allarm Burner" AT %Q6.7 : Bool;   // A 56.2 RESET ALARMBURNER
   "Start High Flame" AT %Q7.0 : Bool;   // A 56.6 START HIGH FLAMEBURNER
   "Foced Spark" AT %Q7.1 : Bool;   // A 56.7 ENABLE SPARK FOR3 sec. DURING
   "103A5" AT %Q7.2 : Bool;
   "103A6" AT %Q7.3 : Bool;
   "103A7" AT %Q7.4 : Bool;
   "Reset_Inverter" AT %Q7.5 : Bool;   // RESET ALARMS INVERTER
   "Siren" AT %Q7.6 : Bool;   // A 57.6 SIREN ALARMS
   "Blinking Ligh" AT %Q7.7 : Bool;   // A 57.7 LAMPALARM
   "EV-11" AT %Q12.0 : Bool;   // A0.0 FILTER 1 VALVE BF01FIRST SECTOR
   "EV-12" AT %Q12.1 : Bool;   // A0.1 FILTER 2 VALVE BF01FIRST SECTOR
   "EV-13" AT %Q12.2 : Bool;   // A0.2 FILTER 3 VALVE BF01FIRST SECTOR
   "EV-14" AT %Q12.3 : Bool;   // A0.3 FILTER 4 VALVE BF01FIRST SECTOR
   "EV-15" AT %Q12.4 : Bool;   // A0.4 FILTER 5 VALVE BF01FIRST SECTOR
   "EV-16" AT %Q12.5 : Bool;   // A0.5 FILTER 6 VALVE BF01FIRST SECTOR
   "EV-17" AT %Q12.6 : Bool;   // A0.6 FILTER 7 VALVE BF01FIRST SECTOR
   "EV-18" AT %Q12.7 : Bool;   // A0.7 FILTER 8 VALVE BF01FIRST SECTOR
   "EV-19" AT %Q13.0 : Bool;   // A1.0 FILTER 1 VALVE BF01SECOND SECTOR
   "EV-20" AT %Q13.1 : Bool;   // A1.1 FILTER 2 VALVE BF01SECOND SECTOR
   "EV-21" AT %Q13.2 : Bool;   // A1.2 FILTER 3 VALVE BF01SECOND SECTOR
   "EV-22" AT %Q13.3 : Bool;   // A1.3 FILTER 4 VALVE BF01SECOND SECTOR
   "EV-23" AT %Q13.4 : Bool;   // A1.4 FILTER 5 VALVE BF01SECOND SECTOR
   "EV-24" AT %Q13.5 : Bool;   // A1.5 FILTER 6 VALVE BF01SECOND SECTOR
   "EV-25" AT %Q13.6 : Bool;   // A1.6 FILTER 7 VALVE BF01SECOND SECTOR
   "EV-26" AT %Q13.7 : Bool;   // A1.7 FILTER 8 VALVE BF01SECOND SECTOR
   "EV-27" AT %Q14.0 : Bool;   // A2.0 FILTER 1 VALVE BF01THIRD SECTOR
   "EV-28" AT %Q14.1 : Bool;   // A2.1 FILTER 2 VALVE BF01THIRD SECTOR
   "EV-29" AT %Q14.2 : Bool;   // A2.2 FILTER 3 VALVE BF01THIRD SECTOR
   "EV-30" AT %Q14.3 : Bool;   // A2.3 FILTER 4 VALVE BF01THIRD SECTOR
   "EV-31" AT %Q14.4 : Bool;   // A2.4 FILTER 5 VALVE BF01THIRD SECTOR
   "EV-32" AT %Q14.5 : Bool;   // A2.5 FILTER 6 VALVE BF01THIRD SECTOR
   "EV-33" AT %Q14.6 : Bool;   // A2.6 FILTER 7 VALVE BF01THIRD SECTOR
   "EV-34" AT %Q14.7 : Bool;   // A2.7 FILTER 8 VALVE BF01THIRD SECTOR
   "EV-35" AT %Q15.0 : Bool;   // A3.0 FILTER 1 VALVE BF01FOURTH SECTOR
   "EV-36" AT %Q15.1 : Bool;   // A3.1 FILTER 2 VALVE BF01FOURTH SECTOR
   "EV-37" AT %Q15.2 : Bool;   // A3.2 FILTER 3 VALVE BF01FOURTH SECTOR
   "EV-38" AT %Q15.3 : Bool;   // A3.3 FILTER 4 VALVE BF01FOURTH SECTOR
   "EV-39" AT %Q15.4 : Bool;   // A3.4 FILTER 5 VALVE BF01FOURTH SECTOR
   "EV-40" AT %Q15.5 : Bool;   // A3.5 FILTER 6 VALVE BF01FOURTH SECTOR
   "EV-41" AT %Q15.6 : Bool;   // A3.6 FILTER 7 VALVE BF01FOURTH SECTOR
   "EV-42" AT %Q15.7 : Bool;   // A3.7 FILTER 8 VALVE BF01FOURTH SECTOR
   "EV-43" AT %Q16.0 : Bool;   // A4.0 FILTER 1 VALVE BF01FIFTH SECTOR
   "EV-44" AT %Q16.1 : Bool;   // A4.1 FILTER 2 VALVE BF01FIFTH SECTOR
   "EV-45" AT %Q16.2 : Bool;   // A4.2 FILTER 3 VALVE BF01FIFTH SECTOR
   "EV-46" AT %Q16.3 : Bool;   // A4.3 FILTER 4 VALVE BF01FIFTH SECTOR
   "EV-47" AT %Q16.4 : Bool;   // A4.4 FILTER 5 VALVE BF01FIFTH SECTOR
   "EV-48" AT %Q16.5 : Bool;   // A4.5 FILTER 6 VALVE BF01FIFTH SECTOR
   "EV-49" AT %Q16.6 : Bool;   // A4.6 FILTER 7 VALVE BF01FIFTH SECTOR
   "EV-50" AT %Q16.7 : Bool;   // A4.7 FILTER 8 VALVE BF01FIFTH SECTOR
   "PV-14" AT %Q17.0 : Bool;   // A 5.0 INLET FRESH AIRFILTERS VALVE
   "Start FN04" AT %Q17.1 : Bool;   // FN-04/FN-04A MOTOR
   "Spare_1" AT %Q17.2 : Bool;   // SPARE
   "Spare_2" AT %Q17.3 : Bool;   // SPARE
   "Spare_3" AT %Q17.4 : Bool;   // SPARE
   "Spare_4" AT %Q17.5 : Bool;   // SPARE
   "Spare_5" AT %Q17.6 : Bool;   // SPARE
   "Spare_6" AT %Q17.7 : Bool;   // SPARE
   "102A5_SPARE0" AT %QW288 : Word;
   "RD01_SP_SPEED" AT %QW290 : Word;   // ROTATING DRUM RD-01
   "FN01_SP_SPEED" AT %QW292 : Word;   // SP SPEED BLOWER FAN FN-01
   "102A5_SPARE3" AT %QW294 : Word;
   "102A5_SPARE4" AT %QW296 : Word;
   "BWF01_SP_FlowRate" AT %QW298 : Word;   // FLOW RATE SPEED SET BWF 01(CLIENT MACHINE)(4-20mA)
   "BWF02_SP_FlowRate" AT %QW300 : Word;   // FLOW RATE SPEED SET BWF 02(CLIENT MACHINE)(4-20mA)
   "LIW_SP_SPEED" AT %QW302 : Word;   // SPEED SET LIW SYSTEM(CLIENT MACHINE)(4-20mA)
   "102A6_SPARE0" AT %QW304 : Word;
   "FN02_SP" AT %QW306 : Word;   // BLOWER FAN FN-02(4-20mA)
   "BR01_GAS_SP" AT %QW308 : Word;   // FLAME MODULATION GAS FLOATING MOTOR BR-01(4-20mA)
   "BR01_AIR_SP" AT %QW310 : Word;   // FLAME MODULATION AIR FLOATING MOTOR BR-01(4-20mA)
   "102A6_SPARE4" AT %QW312 : Word;
   "102A6_SPARE5" AT %QW314 : Word;
   "102A6_SPARE6" AT %QW316 : Word;
   "102A6_SPARE7" AT %QW318 : Word;
   "FN04_SP" AT %QW336 : Word;   // ASPIRATION FAN FN-04 SPEED
   "153A4_SPARE0" AT %QW338 : Word;
   "153A4_SPARE1" AT %QW340 : Word;
   "153A4_SPARE2" AT %QW342 : Word;
   "153A4_SPARE3" AT %QW344 : Word;
   "153A4_SPARE4" AT %QW346 : Word;
   "153A4_SPARE5" AT %QW348 : Word;
   "153A4_SPARE6" AT %QW350 : Word;
END_VAR

TYPE "Tipo Dati 1"
VERSION : 1.0
   STRUCT
      JOB_WR : Struct   // write commands
         NO : Byte;   // number
         BUSY : Bool;   // job in working
         DONE : Bool;   // job is done
         IMPOSS : Bool;   // job impossible
         UNKOWN : Bool;   // job unkown
      END_STRUCT;
      JOB_RD : Struct   // read commands
         NO : Byte;   // number
         BUSY : Bool;   // job in working
         DONE : Bool;   // job is done
         IMPOSS : Bool;   // job impossible
         UNKOWN : Bool;   // job unkown
      END_STRUCT;
      RESERV_0 : Array[1..3] of Word;
      RESERV_1 : Word;   // reserved
      MOD_ADR : Word;   // module address
      CH_ADR : DWord;   // channel address
      DS_OFFS : Byte;   // data block offset
      RESERV_2 : Byte;   // reserved
      CONTROL_SIGNALS : Struct   // control signals
         BIT0_0 : Bool;   // reserved
         BIT0_1 : Bool;   // reserved
         BIT0_2 : Bool;   // reserved
         BIT0_3 : Bool;   // reserved
         BIT0_4 : Bool;   // reserved
         BIT0_5 : Bool;   // reserved
         BIT0_6 : Bool;   // reserved
         BIT0_7 : Bool;   // reserved
         CTRL_DQ0 : Bool;   // control digital output DQ0
         CTRL_DQ1 : Bool;   // control digital output DQ1
         CTRL_DQ2 : Bool;   // control digital output DQ2
         CTRL_DQ3 : Bool;   // control digital output DQ3
         CTRL_DQ4 : Bool;   // control digital output DQ4
         CTRL_DQ5 : Bool;   // control digital output DQ5
         CTRL_DQ6 : Bool;   // control digital output DQ6
         CTRL_DQ7 : Bool;   // control digital output DQ7
         SET_DQ0 : Bool;   // set digital output DQ0
         SET_DQ1 : Bool;   // set digital output DQ1
         SET_DQ2 : Bool;   // set digital output DQ2
         SET_DQ3 : Bool;   // set digital output DQ3
         SET_DQ4 : Bool;   // set digital output DQ4
         SET_DQ5 : Bool;   // set digital output DQ5
         SET_DQ6 : Bool;   // set digital output DQ6
         SET_DQ7 : Bool;   // set digital output DQ7
         SW_GATE0 : Bool;   // software gate 0
         SW_GATE1 : Bool;   // software gate 1
         SW_GATE2 : Bool;   // software gate 2
         SW_GATE3 : Bool;   // software gate 3
         SW_GATE4 : Bool;   // software gate 4
         SW_GATE5 : Bool;   // software gate 5
         SW_GATE6 : Bool;   // software gate 6
         SW_GATE7 : Bool;   // software gate 7
         CTRL_DWORD1 : DWord;   // reserved
         CTRL_DWORD2 : DWord;   // reserved
         CTRL_DWORD3 : DWord;   // reserved
      END_STRUCT;
      CHECKBACK_SIGNALS : Struct   // checkback signals
         BIT0_0 : Bool;   // reserved
         STS_TFB : Bool;   // status test free bit
         BIT0_2 : Bool;   // reserved
         BIT0_3 : Bool;   // reserved
         DATA_ERR : Bool;   // data error bit
         BIT0_5 : Bool;   // reserved
         BIT0_6 : Bool;   // reserved
         PARA : Bool;   // module parametrized
         STS_CMP0 : Bool;   // status compare event 0
         STS_CMP1 : Bool;   // status compare event 1
         STS_CMP2 : Bool;   // status compare event 2
         STS_CMP3 : Bool;   // status compare event 3
         STS_CMP4 : Bool;   // status compare event 4
         STS_CMP5 : Bool;   // status compare event 5
         STS_CMP6 : Bool;   // status compare event 6
         STS_CMP7 : Bool;   // status compare event 7
         STS_UFLW0 : Bool;   // status counter 0 passed the underflow value
         STS_UFLW1 : Bool;   // status counter 1 passed the underflow value
         STS_UFLW2 : Bool;   // status counter 2 passed the underflow value
         STS_UFLW3 : Bool;   // status counter 3 passed the underflow value
         STS_UFLW4 : Bool;   // status counter 4 passed the underflow value
         STS_UFLW5 : Bool;   // status counter 5 passed the underflow value
         STS_UFLW6 : Bool;   // status counter 6 passed the underflow value
         STS_UFLW7 : Bool;   // status counter 7 passed the underflow value
         STS_OFLW0 : Bool;   // status counter 0 passed the overflow value
         STS_OFLW1 : Bool;   // status counter 1 passed the overflow value
         STS_OFLW2 : Bool;   // status counter 2 passed the overflow value
         STS_OFLW3 : Bool;   // status counter 3 passed the overflow value
         STS_OFLW4 : Bool;   // status counter 4 passed the overflow value
         STS_OFLW5 : Bool;   // status counter 5 passed the overflow value
         STS_OFLW6 : Bool;   // status counter 6 passed the overflow value
         STS_OFLW7 : Bool;   // status counter 7 passed the overflow value
         STS_DIR0 : Bool;   // status counter 0 direction
         STS_DIR1 : Bool;   // status counter 1 direction
         STS_DIR2 : Bool;   // status counter 2 direction
         STS_DIR3 : Bool;   // status counter 3 direction
         STS_DIR4 : Bool;   // status counter 4 direction
         STS_DIR5 : Bool;   // status counter 5 direction
         STS_DIR6 : Bool;   // status counter 6 direction
         STS_DIR7 : Bool;   // status counter 7 direction
         STS_DI0 : Bool;   // status of the digital input 0
         STS_DI1 : Bool;   // status of the digital input 1
         STS_DI2 : Bool;   // status of the digital input 2
         STS_DI3 : Bool;   // status of the digital input 3
         STS_DI4 : Bool;   // status of the digital input 4
         STS_DI5 : Bool;   // status of the digital input 5
         STS_DI6 : Bool;   // status of the digital input 6
         STS_DI7 : Bool;   // status of the digital input 7
         STS_DQ0 : Bool;   // status of the digital output 0
         STS_DQ1 : Bool;   // status of the digital output 1
         STS_DQ2 : Bool;   // status of the digital output 2
         STS_DQ3 : Bool;   // status of the digital output 3
         STS_DQ4 : Bool;   // status of the digital output 4
         STS_DQ5 : Bool;   // status of the digital output 5
         STS_DQ6 : Bool;   // status of the digital output 6
         STS_DQ7 : Bool;   // status of the digital output 7
         STS_GATE0 : Bool;   // status of the internal gate 0
         STS_GATE1 : Bool;   // status of the internal gate 1
         STS_GATE2 : Bool;   // status of the internal gate 2
         STS_GATE3 : Bool;   // status of the internal gate 3
         STS_GATE4 : Bool;   // status of the internal gate 4
         STS_GATE5 : Bool;   // status of the internal gate 5
         STS_GATE6 : Bool;   // status of the internal gate 6
         STS_GATE7 : Bool;   // status of the internal gate 7
         USER_STAT_WORD0 : Word;   // user specific status
         USER_STAT_WORD1 : Word;   // user specific status
         USER_STAT_WORD2 : Word;   // user specific status
         USER_STAT_WORD3 : Word;   // user specific status
      END_STRUCT;
      LOAD_VAL0 : DInt;   // load value counter 0
      LOAD_VAL1 : DInt;   // load value counter 1
      LOAD_VAL2 : DInt;   // load value counter 2
      LOAD_VAL3 : DInt;   // load value counter 3
      LOAD_VAL4 : DInt;   // load value counter 4
      LOAD_VAL5 : DInt;   // load value counter 5
      LOAD_VAL6 : DInt;   // load value counter 6
      LOAD_VAL7 : DInt;   // load value counter 7
      LOAD_PREPARE_VAL0 : DInt;   // load prepare value counter 0
      LOAD_PREPARE_VAL1 : DInt;   // load prepare value counter 1
      LOAD_PREPARE_VAL2 : DInt;   // load prepare value counter 2
      LOAD_PREPARE_VAL3 : DInt;   // load prepare value counter 3
      LOAD_PREPARE_VAL4 : DInt;   // load prepare value counter 4
      LOAD_PREPARE_VAL5 : DInt;   // load prepare value counter 5
      LOAD_PREPARE_VAL6 : DInt;   // load prepare value counter 6
      LOAD_PREPARE_VAL7 : DInt;   // load prepare value counter 7
      CMP_VAL0 : DInt;   // comparator value 0
      CMP_VAL1 : DInt;   // comparator value 1
      CMP_VAL2 : DInt;   // comparator value 2
      CMP_VAL3 : DInt;   // comparator value 3
      CMP_VAL4 : DInt;   // comparator value 4
      CMP_VAL5 : DInt;   // comparator value 5
      CMP_VAL6 : DInt;   // comparator value 6
      CMP_VAL7 : DInt;   // comparator value 7
      ACT_CNTV0 : DInt;   // actual counter value 0
      ACT_MSRV0 : DInt;   // act. measurement value 0
      ACT_CNTV1 : DInt;   // actual counter value 1
      ACT_MSRV1 : DInt;   // act. measurement value 1
      ACT_CNTV2 : DInt;   // actual counter value 2
      ACT_MSRV2 : DInt;   // act. measurement value 2
      ACT_CNTV3 : DInt;   // actual counter value 3
      ACT_MSRV3 : DInt;   // act. measurement value 3
      ACT_CNTV4 : DInt;   // actual counter value 4
      ACT_MSRV4 : DInt;   // act. measurement value 4
      ACT_CNTV5 : DInt;   // actual counter value 5
      ACT_MSRV5 : DInt;   // act. measurement value 5
      ACT_CNTV6 : DInt;   // actual counter value 6
      ACT_MSRV6 : DInt;   // act. measurement value 6
      ACT_CNTV7 : DInt;   // actual counter value 7
      ACT_MSRV7 : DInt;   // act. measurement value 7
      DIAGNOSTIC_INT_INFO : Struct   // diagnostic int. information
         BYTE0 : Byte;   // byte 0
         BYTE1 : Byte;   // byte 1
         BYTE2 : Byte;   // byte 2
         BYTE3 : Byte;   // byte 3
         BYTE4 : Byte;   // channel type info
         BYTE5 : Byte;   // channel info length
         BYTE6 : Byte;   // number of channels
         BYTE7 : Byte;   // channel error vector
         BYTE8 : Byte;   // error counter 0
         BYTE9 : Byte;   // error counter 1
         BYTE10 : Byte;   // error counter 2
         BYTE11 : Byte;   // error counter 3
         BYTE12 : Byte;   // error counter 4
         BYTE13 : Byte;   // error counter 5
         BYTE14 : Byte;   // error counter 6
         BYTE15 : Byte;   // error counter 7
      END_STRUCT;
   END_STRUCT;
END_TYPE

TYPE "Motor"
   STRUCT
      Risposta : Bool;
      Allarme_comulativo : Bool;
   END_STRUCT;
END_TYPE

TYPE "Motorized Valve"
   STRUCT
      Risposta_opening : Bool;
      Risposta_closing : Bool;
      Comulativo_allarmi : Bool;
      Limit_switch_open : Bool;
      Limit_switch_close : Bool;
   END_STRUCT;
END_TYPE

TYPE "Valve"
   STRUCT
      LS_Open : Bool;
      LS_Close : Bool;
      Total_allarms : Bool;
   END_STRUCT;
END_TYPE

TYPE "Client Motor"
   STRUCT
      Status : Bool;
      Risposta : Bool;
      Allarme_Comulativo : Bool;
      Livello_Max : Bool;
      Livello_Min : Bool;
   END_STRUCT;
END_TYPE

TYPE "PV_1_GATE"
   STRUCT
      LS_Open : Bool;
      LS_Close : Bool;
      Selector : Bool;
      Total_Allarms : Bool;
   END_STRUCT;
END_TYPE

TYPE "PV_2_GATE"
   STRUCT
      Comulativo_Allarmi : Bool;
      LS_Gate_A_Open : Bool;
      LS_Gate_A_Close : Bool;
      LS_Gate_B_Open : Bool;
      LS_Gate_B_Close : Bool;
      Selector_GateA : Bool;
      Selector_GateB : Bool;
   END_STRUCT;
END_TYPE

TYPE "Recipe"
   STRUCT
      BWF01 : Int;   // Scraps Feeder 1 - %
      BWF02 : Int;   // Scraps Feeder 2 - %
      RD01 : Int;   // Rotary Drum Speed - %
      FN01 : Int;   // Blower Fan Speed - %
      PSH01 : Int;   // Secondary Line Air Pressure HMI Resc - mb
      PSH02 : Int;   // Decoating line MAX air pressure HMI Resc - mb
      TC03 : Int;   // Decoating Temperature - °C
      TC01 : Int;   // AfterBurner Temperature - °C
      Spare : Word;   // Spare data
      Spare_1 : Word;   // Spare data
      Spare_2 : Word;   // Spare data
   END_STRUCT;
END_TYPE

TYPE "BR-01"
   STRUCT
      High_Flame : Bool;
      Burner_on : Bool;
   END_STRUCT;
END_TYPE

DATA_BLOCK "Data"   // DB1
{ S7_Optimized_Access := 'FALSE' }
VERSION : 0.1
   VAR
      SET_PERC_BWF01 : Int := 30;   // (SET_PERC_TR01)
      SET_PERC_BWF02 : Int := 40;   // (SET_PERC_VT00)
      Set_Perc_VT02 : Int := 35;   // Set speed FN02
      SET_PERC_FR01 : Int := 55;   // (SET_PERC_FR01)
      SET_PERC_VT01 : Int := 64;   // (SET_PERC_VT01)
      SET_PERC_FN04 : Int := 80;   // (SET_PERC_TM01)
      TC06 : Int := 0;   // (TC06)
      SET_PERC_VT4 : Int := 0;   // (SET_PERC_VT4)
      SET_EVR1A_Open_time : Word := 16#0400;   // (SET_EVR1A_Open_time)
      Burner_Air_Out : Int := 35;   // (SET_PERC_BURNER)
      RO01_SETPOINT : Int := 0;   // (RO01_SETPOINT_MIN)
      Burner_Panel_SetPoint : Int := 35;   // (RO01_SETPOINT_MAX)
      PSH03 : Int := -10;
      RO01_MAX_SETPOINT : Int := 100;
      PSH02_MAX_SETPOINT : Int := 3;
      PC01_S000000000 : Int := 0;   // (PC01_SETPOINT_MIN)
      PSH01_SETPOINT : Int := 20;   // (PC01_SETPOINT_MAX)
      Free_34 : Int := 0;
      Free_36 : Int := 0;
      Free_38 : Int := 0;
      PSH03_SETPOINT : Int := 10;   // (PC02_SETPOINT_MIN)
      PSH02_SETPOINT : Int := 0;   // (PC02_SETPOINT_MAX)
      SET_EVR1B_Open_time : Word := 16#0400;
      PV04_Clean_Delay : Word := 16#1600;   // (PC02_PULSE_TIME)
      PC02_KP0000000 : Int := 0;   // (PC02_KP)
      TC03_SETPOINT : Int := 450;   // (TC03_SETPOINT_MIN)
      Free_52 : Int := 0;
      TC09_MAX : Int := 180;
      TC09_MAX_MAX : Int := 200;
      Free_58 : Int := 0;
      Free_60 : Int := 0;
      TC00030_V0000000 : Int := 0;   // (TC03_VG1_KP)
      RO03 : Int := 0;   // (RO03)
      TC01_SETPOINT : Int := 660;   // (TC01_SETPOINT)
      TC01_MAX_ALL : Int := 1200;   // (TC01_MAX_ALL)
      Free_70 : Int := 0;   // (TC01_MAX_MAX_ALL)
      TC03_MIN_ALL : Int := 400;   // (TC03_MIN_ALL)
      TC03_MAX_ALL : Int := 750;   // (TC03_MAX_ALL)
      Free_76 : Int := 0;   // (TC03_MAX_MAX_ALL)
      RO04 : Int := -9999;   // (RO04)
      Min_Pressure_PC_01 : Int := -10;   // (T3_MAX_ALL)
      Free_82 : Int := 0;   // (T3_MAX_MAX_ALL)
      TC04_TC05_MAX_ALL : Int := 120;   // (TC04_TC05_MAX_ALL)
      Free_86 : Int := 0;   // (T5_T6_MAX_ALL)
      SIREN_WORK_TIME : S5Time := S5T#20S;   // (SIREN_WORK_TIME)
      D37 : Int := 2;   // (D37)
      EVFR01_Work_time : Word := 16#0700;   // (EVFR01_Work_time)
      EVFR01_Wait_time : Word := 16#2400;   // (EVFR01_Wait_time)
      Tempo_presetting : Int := 0;   // (Time_presetting)
      Tipo_preset : Int := 2;   // (Type_preset)
      Amp_RD01 : Int := 27;   // (Amp_FR01)
      Amp_FN01 : Int := 71;   // (Amp_VT01)
      Amp_FN040000000 : Int := 0;
      Amp_VT0300000000 : Int := 0;   // (Amp_VT03)
      Temp_TC02 : Int := 656;   // (Temp_TC02)
      Temp_TC01 : Int := 664;   // (Temp_TC01)
      Temp_TC03 : Int := 482;   // (Temp_TC03)
      Temp_T3000000000 : Int := 0;   // (Temp_T3)
      Temp_TC04 : Int := 4;   // (Temp_TC04)
      Temp_TC05 : Int := -9999;   // (Temp_TC05)
      Temp_T6 : Int := 450;   // (Temp_T6)
      Pot00000000000009 : Int := 0;   // (Pot_BR1)
      Max_PRC_BR1 : Int := 45;   // (Max_PRC_BR1)
      DP_ASPI00000000000000 : Int := 100;   // (DP_ASPIR_PC03)
      Oxigen_RO02 : Int := -9999;   // (Oxigen_RO02)
      Oxigen_RO01 : Int := -9999;   // (Oxigen_RO01)
      Gas00000000000000 : Int := 0;   // (GasM)
      Press_PC01 : Int := -1;   // (Press_PC01)
      Pot_MV06 : Int := 0;   // (Press_PC02)
      Pot_MV04A : Int := 0;   // (Free_138)
      Pot_MV05 : Int := 0;   // (Pot_MV01)
      Pot_MV02 : Int := 0;   // (Pot_MV02)
      Pot_MV03 : Int := 55;   // (Pot_MV03)
      Pot_MV04B : Int := 0;   // (Pot_MV04)
      Pot_MV01 : Int := 100;   // (Pot_VG01)
      LD_01V_WorkTime : Word := 16#0300;   // (VB01_Work_Time)
      LD_01V_PauseTime : Word := 16#2120;   // (VB01_Pause_Time)
      SET_PV02B_Open_time : Word := 16#0200;
      SET_PV02A_Open_time : Word := 16#0200;
      Free158 : S5Time := S5T#0MS;   // (EV01_Work_Time)
      Free160 : S5Time := S5T#0MS;   // (EV01_Pause_Time)
      Free162 : S5Time := S5T#0MS;   // (EVSA_Work_Time)
      Free164 : S5Time := S5T#0MS;   // (EVSA_Pause_Time)
      Free166 : S5Time := S5T#0MS;   // (FREE_W166)
      Free168 : S5Time := S5T#0MS;   // (FREE_W168)
      Ev_filter_on : Int := 25;
      TC_040000000 : Int := 0;
      TC_0500000 : Int := 0;
      CLIENT_1 : Int := 3;
      CLIENT_2 : Int := 13;
      CLIENT_3 : Int := -9999;
      TC_01 : Int := 0;
      TC_02 : Int := 0;
      TC_03 : Int := 0;
      TC_06 : Int := 0;
      TC_07 : Int := -9999;
      ZT_01 : Int := -9999;
      PSH_01 : Int := 0;
      PSH_02 : Int := 0;
      RO_01 : Int := 0;
      RO_02 : Int := 0;
      RO_03 : Int := 0;
      RO_04 : Int := 0;
      GAS_BR_01 : Int := 63;
      AIR_BR_01 : Int := 32;
      MASSICO_FLOW_GAS : Int := 168;
      MASSICO_FLOW_AIR : Int := 1599;
      MV_05 : Int := 0;
      MV_02 : Int := 0;
      MV_06 : Int := 0;
      MV_04 : Int := 0;
      FN_02_FAN : Int := 34;
      FN_04_ASPIRATOR : Int := 97;
      RD_01 : Int := 0;
      FN_01 : Int := 0;
      LAVA : Int := 0;
      LAVA_START : Int := 11;
      LAVA_END : Int := 90;
      LAVA_PAUSA : Word := 16#0400;
      LAVA_LAVORO : Word := 16#0020;
      DP_01 : Int := 29;
      DP_02 : Int := 140;
      PC_01 : Int := -44;
      SET_POS_MV05 : Int := 0;
      SET_POS_MV02 : Int := 100;
      SET_POS_MV04 : Int := 100;
      Burner_Gas_Out : Int := 71;
      ENCODER_MV03 : Int := 0;
      ENCODER_MV01 : Int := 0;
      CLIENT_4 : Int := 69;
      P0000000000 : Int := 0;
      TC_09 : Int := 61;
      TC_10 : Int := -9999;
      BWF01_count : Int := 10;
      BWF02_count : Int := 1;
      BWF01_count_rep : Int := 0;
      BWF02_count_rep : Int := 0;
      Free_04 : Int := 0;
      Free_05 : Int := 0;
      Free_06 : Int := 0;
      Free_07 : Int := 0;
      Free_08 : Int := 0;
      Free_09 : Int := 0;
      Maint_code_0 : Int := 1;
      Maint_code_1 : Int := 1;
      Maint_code_3 : Int := 1;
      Free_013 : Int := 0;
      Free_014 : Int := 0;
      Free_015 : Int := 0;
      Free_016 : Int := 0;
      "PV-01a" : Int := 40;
      PV_01B : Int := 40;
      PV_02A : Int := 20;
      PV_02B : Int := 20;
      LD01_W : Int := 30;
      LD01_P : Int := 1200;
      EV_03_W : Int := 70;
      EV_03P : Int := 4000;
      PV04 : Int := 600;
      VALVE_W : Int := 2;
      VALVE_P : Int := 40;
      Siren_time : Int := 200;
   END_VAR
BEGIN
END_DATA_BLOCK

DATA_BLOCK "Flag"   // DB2
{ S7_Optimized_Access := 'FALSE' }
VERSION : 0.1
   VAR
      M_BC_01 : Bool;   // COM_W0 BIT8 (M_TR01)
      M_RD_01 : Bool;   // COM_W0 BIT9 (M_MN02)
      M_RD_01_FAN : Bool;   // COM_W0 BIT10 (M_MR1)
      M_MC_03 : Bool;   // COM_W0 BIT11 (M_VT00_CLIENTE)
      M_MC_04 : Bool;   // COM_W0 BIT12 (M_VB01)
      M_MC_05 : Bool;   // COM_W0 BIT13 (M_FR01)
      M_VS_01 : Bool;   // COM_W0 BIT14 (M_Servo_FR01)
      M_SC_12 : Bool;   // COM_W0 BIT15 (M_MN03)
      M_FN_02 : Bool;   // COM_W0 BIT0 (M_VV01AB)
      M_VR_01 : Bool;   // COM_W0 BIT1 (M_TM01)
      M_FN_01 : Bool;   // COM_W0 BIT2 (M_MN04)
      M_VR_02 : Bool;   // COM_W0 BIT3 (M_MBN4_SX00000)
      M_CH_01 : Bool;   // COM_W0 BIT4 (M_MBN4_DX00000)
      M_FN_03 : Bool;   // COM_W0 BIT5 (M_VA01AB)
      M_SC_01 : Bool;   // COM_W0 BIT6 (M_VT01)
      M_FN_01_FAN : Bool;   // COM_W0 BIT7 (M_VR03)
      M_LD_01 : Bool;   // COM_W1 BIT8 (M_VT00_AUTO)
      M_LD_01_VIB : Bool;   // COM_W1 BIT9 (M_MV01_Open)
      M_SC_10 : Bool;   // COM_W1 BIT10 (M_MV01_Close)
      M_SC_11 : Bool;   // COM_W1 BIT11 (M_MV01_Close)
      M_FN_04 : Bool;   // COM_W1 BIT12 (M_MV02_Close)
      M_VR_03 : Bool;   // COM_W1 BIT13 (M_MV03_Open)
      M_VR_04 : Bool;   // COM_W1 BIT14 (M_MV03_Close)
      M_VR_05 : Bool;   // COM_W1 BIT15 (M_MCV500000000)
      M_VR_06 : Bool;   // COM_W1 BIT0 (M_TSHL0000000)
      M_FN_05 : Bool;   // COM_W1 BIT1 (M_MV04_Open)
      SPARE : Bool;   // COM_W1 BIT2 (M_MV04_Close)
      M_MV01_OPEN : Bool;   // COM_W1 BIT3 (M_VG01_Open)
      M_MV01_Close : Bool;   // COM_W1 BIT4 (M_VG01_Close)
      M_Aux_INV : Bool;   // COM_W1 BIT5 (M_SERVO_VT01)
      SPARE_2 : Bool;   // COM_W1 BIT6 (M_MVT02)
      M_FN_06 : Bool;   // COM_W1 BIT7 (M_CH01)
      SPARE_3 : Bool;   // COM_W2 BIT8 (M_VT03)
      M_PV04 : Bool;   // COM_W2 BIT9 (BURNER_OPEN)
      SPARE_4 : Bool;   // COM_W2 BIT10 (BURNER_CLOSE)
      AUTO_BURNER : Bool;   // COM_W2 BIT11 (AUTO_BURNER)
      SPARE_5 : Bool;   // COM_W2 BIT12 (M_VR01)
      SPARE_6 : Bool;   // COM_W2 BIT13 (M_VR02)
      SPARE_7 : Bool;   // COM_W2 BIT14 (GROUND_MODE)
      R1_GATE_LOOP_ON : Bool;   // COM_W2 BIT15 (R1_GATE_LOOP_ON)
      Enable_R1_GATE : Bool;   // COM_W2 BIT0 (Disable_R1_GATE)
      Burner_ready : Bool;   // COM_W2 BIT1 (Burner_ready)
      Start_Burner : Bool;   // COM_W2 BIT2 (Start_Burner)
      SPARE_8 : Bool;   // COM_W2 BIT3 (M_SERVO_VT02)
      M_ER01 : Bool;   // COM_W2 BIT4 (M_MRT300000000)
      SPARE_9 : Bool;   // COM_W2 BIT5 (M_MVV2000000000)
      SPARE_10 : Bool;   // COM_W2 BIT6 (M_DM01000000000)
      SPARE_11 : Bool;   // COM_W2 BIT7 (B047)
      RESET_ALLARM : Bool;   // COM_W3 BIT8 (RESET_ALLARM)
      RUN_HORN : Bool;   // COM_W3 BIT9 (RUN_HORN)
      STOP_HORN : Bool;   // COM_W3 BIT10 (STOP_HORN)
      NEW_ALLARM : Bool;   // COM_W3 BIT11 (NEW_ALLARM)
      M_HORN : Bool;   // COM_W3 BIT12 (M_HORN)
      MV06_Auto : Bool;   // COM_W3 BIT13 (B053)
      MV05_Auto : Bool := TRUE;   // COM_W3 BIT14 (MV01_Auto)
      MV02_Auto : Bool := TRUE;   // COM_W3 BIT15 (MV02_Auto)
      MV03_Auto : Bool := TRUE;   // COM_W3 BIT0 (MV03_Auto)
      MV04_Auto : Bool := TRUE;   // COM_W3 BIT1 (MV04_Auto)
      MV01_Auto : Bool := TRUE;   // COM_W3 BIT2 (VG01_Auto)
      Auto_ON1 : Bool;   // COM_W3 BIT3 (Auto_ON1)
      STANDBY_ON : Bool;   // COM_W3 BIT4 (STANDBY_ON)
      Maintenance_ON : Bool;   // COM_W3 BIT5 (Auto_OFF1)
      SPARE_12 : Bool;   // COM_W3 BIT6 (B062)
      M_TDPRO_REPORT : Bool;   // COM_W3 BIT7 (M_TDPRO_REPORT)
      PV_01_GATE_A_MEM_CLOSE : Bool := TRUE;
      PV_01_GATE_A_MEM_OPEN : Bool;
      PV_01_GATE_B_MEM_CLOSE : Bool := TRUE;
      PV_01_GATE_B_MEM_OPEN : Bool;
      PV_02_GATE_A_MEM_CLOSE : Bool := TRUE;
      PV_02_GATE_A_MEM_OPEN : Bool;
      PV_02_GATE_B_MEM_CLOSE : Bool := TRUE;
      PV_02_GATE_B_MEM_OPEN : Bool;
      PV_03_GATE_MEM_CLOSE : Bool;
      PV_03_GATE_MEM_OPEN : Bool := TRUE;
      FN_04_AUTO : Bool;
      M_MV05_CLOSE : Bool;
      M_MV05_OPEN : Bool;
      M_MV02_CLOSE : Bool;
      M_MV02_OPEN : Bool;
      M_MV03_OPEN : Bool;
      M_MV03_CLOSE : Bool;
      M_MV04_OPEN : Bool;
      M_MV04_CLOSE : Bool;
      Enable_R2_GATE : Bool;
      R2_GATE_LOOP_ON : Bool;
      MV06_Open : Bool;
      MV06_Close : Bool;
      SPARE_13 : Bool;
      SPARE_14 : Bool;
      SPARE_15 : Bool;
      M_PV03 : Bool := TRUE;
      SPARE_16 : Bool;
      SPARE_17 : Bool;
      SPARE_18 : Bool;
      SPARE_19 : Bool;
      SPARE_20 : Bool;
      M_BWF01 : Bool;
      SPARE_21 : Bool;
      SPARE_22 : Bool;
      SPARE_23 : Bool;
      SPARE_24 : Bool;
      M_BWF02 : Bool;
      SPARE_25 : Bool;
      SPARE_26 : Bool;
      SPARE_27 : Bool;
      M_PV14 : Bool;
      MV04_Close : Bool;
      MV04_Open : Bool;
      Reset_Allarms_HMI : Bool;
      Stop_horn_HMI : Bool;
      SPARE_30 : Bool;
      SPARE_31 : Bool;
      SPARE_32 : Bool;
      SPARE_33 : Bool;
      SPARE_34 : Bool;
      SPARE_35 : Bool;
      SPARE_36 : Bool;
      SPARE_37 : Bool;
      SPARE_38 : Bool;
      SPARE_39 : Bool;
      SPARE_40 : Bool;
      SPARE_41 : Bool;
      SPARE_42 : Bool;
      SPARE_43 : Bool;
      SPARE_44 : Bool;
      SPARE_45 : Bool;
      SPARE_46 : Bool;
      SPARE_47 : Bool;
      SPARE_48 : Bool;
   END_VAR
BEGIN
END_DATA_BLOCK

DATA_BLOCK "Allarm"   // DB3
{ S7_Optimized_Access := 'FALSE' }
VERSION : 0.1
   VAR
      BC_01_FAULT : Bool;   // 0 (TR01_FAULT) / [db3.dbx0.0] BC-01 belt FAULT
      RD_01_FAULT : Bool;   // 1 (LSTR01_FAULT) / RD-01 Rotary drum FAULT
      RD_01_FAN_FAULT : Bool;   // 2 (VTR1_FAULT) / RD-01 Rotary drum fan FAULT
      MC_03_FAULT : Bool;   // 3 (MN02_FAULT) / MC-03 FAULT
      MC_04_FAULT : Bool;   // 4 (LSMN02_FAULT) / MC-04 Metallic conveyor FAULT
      MC_05_FAULT : Bool;   // 5 (ZSXMN02_FAULT) / MC-05 Metallic conveyor FAULT
      VS_01_FAULT : Bool;   // 6 (LOW_TC06_TEMP) / VS-01 Vibrating screen FAULT
      SC_12_FAULT : Bool;   // 7 (GateA_NOT_OPEN) / SC-12 Dust discharge screw FAULT
      FN_02_FAULT : Bool;   // 8 (GateA_NOT_CLOSE) / FN-02 Secondary line fan FAULT
      VR_01_FAULT : Bool;   // 9 (GateB_NOT_OPEN) / VR-01 Cyclon 1 rotary valve FAULT
      FN_01_FAULT : Bool;   // 10 (GateB_NOT_CLOSE) / FN-01 Primary line fan FAULT
      VR_02_FAULT : Bool;   // 11 (FR01_FAULT) / VR-02 Cyclon 3 rotary valve FAULT
      CH_01_FAULT : Bool;   // 12 (SERVO_FR01_FAULT) / CH-01 Chiller FAULT
      FN_03_FAULT : Bool;   // 13 (MN03_FAULT) / FN-03 Burner fan FAULT
      SC_01_FAULT : Bool;   // 14 (LSMN03_FAULT) / SC-01 Cyclon 2/4/5 screw FAULT
      FN_01_FAN_FAULT : Bool;   // 15 (ZSXMN03_FAULT) / FN-01 Primary line fan cooling motor FAULT
      LD_01_FAULT : Bool;   // 16 (VV01AB_FAULT) / LD-01 lime dosator FAULT
      LD_01_VIB_FAULT : Bool;   // 17 (TM01_FAULT) / LD-01-VIB lime vibrator FAULT
      SC_10_FAULT : Bool;   // 18 (MN04_FAULT) / SC-10 Filter 1 screw FAULT
      SC_11_FAULT : Bool;   // 19 (LSMN04_FAULT) / SC-11 Filter 2 screw FAULT
      FN_04_FAULT : Bool;   // 20 (ZSXMN04_FAULT) / FN-04 Primary aspirator FAULT
      VR_03_FAULT : Bool;   // 21 (MBN04_FAULT) / VR-03 cyclon 2/4/5 rotary valveFAULT
      VR_04_FAULT : Bool;   // 22 (VA02AB_FAULT) / VR-04 Filter 1 rotary valve FAULT
      VR_05_FAULT : Bool;   // 23 (VT01_FAULT) / VR-05 Filter 2 rotary valve FAULT
      VR_06_FAULT : Bool;   // 24 (MVT2_FAULT) / VR-06 lime rotoary valve FAULT
      FN_05_FAULT : Bool;   // 25 (VT02_FAULT) / FN-05 Lime fan FAULT
      BC_01_FC : Bool;   // 26 (VR03_FAULT) / BC-01 Trip wire limit switch
      BC_01_PROXIMITY : Bool;   // 27 (MV01_FAULT) / BC-01 Proximity sensor
      MC_03_TORQUE : Bool;   // 28 (SERVOVT01_FAULT) / MC-03 Torque limit switch
      MC_04_TORQUE : Bool;   // 29 (CH01_FAULT) / MC-04 Torque limit switch
      MC_05_TORQUE : Bool;   // 30 (VB01_Fault) / MC-05 Torque limit switch
      MBVA01_FAULT : Bool;   // 31 (MBVA01_FAULT) / FN-06 fan FAULT
      MV02_FAULT : Bool;   // 32 (MV02_FAULT) / MV-02 Motorized valve fault
      VR01_FAULT00000000000000 : Bool;   // 33 (VR01_FAULT) / 4.1
      VR02_FAULT00000000000000 : Bool;   // 34 (VR02_FAULT) / [db3.dbx4.2]
      MV03_FAULT : Bool;   // 35 (MV03_FAULT) / MV-03 Motorized valve FAULT
      RO01_Signal_Fault : Bool;   // 36 (RO01_Signal_Fault) / RO01-RO02 Signal compare FAULT
      Low_Aspiration : Bool;   // 37 (PSL04_FAULT) / PC-01 Low depressure
      PV04_FAULT : Bool;   // 38 (CV5_NOT_OPEN0000) / PV-04 Discharge drum chamber FAULT
      MV01_FAULT : Bool;   // 39 (VG01_FAULT) / MV-01 Motorized valve fault
      RO03_Min : Bool;   // 40 (MCLF_FAULT0000) / Oxygen RO03 too low
      RO03_Max : Bool;   // 41 (ZXMCLF_FAULT) / Oxygen RO03
      MR3_FAULT00000 : Bool;   // 42 (MR3_FAULT00000) / [db3.dbx5.2]
      ZXTR01_FAULT0000000000 : Bool;   // 43 (ZXTR01_FAULT) / [db3.dbx5.3]
      PSL_AIR_LOW : Bool;   // 44 (PSL_AIR_LOW) / PSL-04 Low air pressure
      MV04_FAULT : Bool;   // 45 (MV04_FAULT) / MV-04 Motorized valve FAULT
      VT00_FAULT00000000000 : Bool;   // 46 (VT00_FAULT) / [db3.dbx5.6]
      LD_01_MIN : Bool;   // 47 / LD-01 Low lime level
      FN03_Fault : Bool;   // 48 (MVT04_FAULT) / FN-03 Burner fan FAULT
      SERVOVT02_FAULT0000000 : Bool;   // 49 (SERVOVT02_FAULT) / [db3.dbx6.1]
      VT1_B0000000000000 : Bool;   // 50 (VT1_Bearing_A_Fault) / [db3.dbx6.2]
      VT1_Bea0000 : Bool;   // 51 (VT1_Bearing_B_Fault) / [db3.dbx6.3]
      LOW_GAS_PRESS00000 : Bool;   // 52 (LOW_GAS_PRESS00000) / [db3.dbx6.4
      HIGH_GAS_PRESS00000 : Bool;   // 53 (HIGH_GAS_PRESS00000) / [db3.dbx6.5]
      LOW_BUR000000000 : Bool;   // 54 (LOW_BURNER_AIR_PRESS) / [db3.dbx6.6]
      BURNER_START_FAULT : Bool;   // 55 (BURNER_START_FAULT) / [db3.dbx6.7] Burner start fault
      SERVOMOTOR_MIN_POS_ALL : Bool;   // 56 (SERVOMOTOR_MIN_POS_ALL) / Burner servomotor not in minimal position
      HYDROGEN_BOX_FAULT : Bool;   // 57 (HYDROGEN_BOX_FAULT) / Hydrogen box not ready
      Sechio_Limits : Bool;   // 58 (PV7_FAULT00000) / Stoichiometry out of range
      PV8_FAULT00000 : Bool;   // 59 (PV8_FAULT00000) / [db3.dbx7.3]
      BURNER_LDU_FAULT : Bool;   // 60 (BURNER_LDU_FAULT) / Burner control box FAULT
      Maintenance_ON : Bool;   // 61 (GH1_NOT_OPEN0000) / Maintenence mode !!!!
      MAINTENANCE_PERIOD_LIMIT : Bool;   // MAINTENANCE PERIOD LIMITS
      BURNER_TIME_LIMIT_22H : Bool;   // 63 (MVV2_FAULT00000) / Burner continuous working time limit
      MAX_TC01_TEMP : Bool;   // 64 (MAX_TC01_TEMP) / MAX TC01 temperature
      MAX_MAX_TC01_TEMP : Bool;   // 65 (MAX_MAX_TC01_TEMP) / Extremely high TC01 temperature
      MAX_PSH_02 : Bool;   // 66 (MAX_T5_T6_TEMP00000) / Max pressure PSH-02
      LOW_TC03_TEMP : Bool;   // 67 (LOW_TC03_TEMP) / Low TC03 temperature
      MAX_TC03_TEMP : Bool;   // 68 (MAX_TC03_TEMP) / MAX TC03 temperature
      MAX_MAX_TC03_TEMP : Bool;   // 69 (MAX_MAX_TC03_TEMP) / Extremely high TC03 temperature
      MAX_TC09 : Bool;   // High TC-09 filter temperature
      MAX_MAX_TC09 : Bool;   // Extremly high TC-09 filter temperature
      ZT01_FN01_Vibration : Bool;   // High vibrations FN-01
      TC01_TC02_COMP_FAULT : Bool;   // 73 (TC01_TC02_COMP_FAULT) / TC01/TC02 signal compare fault
      MAX_TC04_TEMP : Bool;   // 74 (MAX_TC04_TEMP) / MAX TC04 temperature
      MAX_TC05_TEMP : Bool;   // 75 (MAX_TC05_TEMP) / MAX TC05 temperature
      Oxigen_LOW : Bool;   // 76 (Oxigen_LOW) / RO01 Oxigen low limit
      MAX_DP_FILTER : Bool;   // 77 (MAX_DP_FILTER0000) / Max filter depressure
      Oxigen_Fault : Bool;   // 78 (Oxigen_Fault) / Oxigen analyzer out of range
      Oxigen_Too_high : Bool;   // 79 (LSL_Low_Level) / Oxigen too high
      anomaly_burner : Bool;   // 10.0
      PV_01_GATE_A_NOT_OPEN : Bool;   // PV-01 Gate A not open
      PV_01_GATE_A_NOT_CLOSE : Bool;   // PV-01 Gate A not close
      PV_01_GATE_B_NOT_OPEN : Bool;   // PV-01 Gate B not open
      PV_01_GATE_B_NOT_CLOSE : Bool;   // PV-01 Gate B not close
      PV_02_GATE_A_NOT_OPEN : Bool;   // PV-02 Gate A not open
      PV_02_GATE_A_NOT_CLOSE : Bool;   // PV-02 Gate A not close
      PV_02_GATE_B_NOT_OPEN : Bool;   // PV-02 Gate B not open
      PV_02_GATE_B_NOT_CLOSE : Bool;   // PV-02 Gate B not close
      PV_03_GATE_NOT_OPEN1 : Bool;   // PV-03 not open
      PV_03_GATE_NOT_CLOSE1 : Bool;   // PV-03 not close
      MV_03_FAULT : Bool;   // MV-03 Motorized valve FAULT
      "110V_Fault" : Bool;   // No 110V Voltage
      MV_05_FAULT : Bool;   // MV-05 Motorized valve FAULT
      MV_06_FAULT : Bool;   // MV-06 Motorized valve FAULT
      BWF01_FAULT : Bool;   // BWF 01 Scraps feeder FAULT
      BWF01_min_LEVEL : Bool;   // BWF 01 Min level
      BWF01_MAX_LEVEL : Bool;   // BWF 01 MAX level
      BWF01_FREE01 : Bool;   // [db3.dbx12.2]
      BWF01_FREE02 : Bool;   // [db3.dbx12.3]
      BWF02_FAULT : Bool;   // BWF 02 Scraps feeder FAULT
      BWF02_min_LEVEL : Bool;   // BWF 02 Min level
      BWF02_MAX_LEVEL : Bool;   // BWF 02 MAX level
      Formula_Fault : Bool;   // Incorrect scraps feeder formula
      BWF02_FREE02 : Bool;   // [db3.dbx13.0]
      BWF01_MAX_LEVEL1 : Bool;   // [db3.dbx13.1]
      BWF01_FREE011 : Bool;   // [db3.dbx13.2]
      BWF01_FREE021 : Bool;   // [db3.dbx13.3]
      Fault_PV14 : Bool;   // PV-14 cold air filter FAULT
      Fault_PV15 : Bool;   // [db3.dbx13.5]
      Fault_PV16 : Bool;   // [db3.dbx13.6]
      Fault_PV17 : Bool;   // [db3.dbx13.7]
      Fault_PV18 : Bool;   // [db3.dbx14.0]
      motor_client_01_fault : Bool;   // Apron conveyor fault (CL01)
      motor_client_02_fault : Bool;   // Impactor fault (CL02)
      motor_client_03_fault : Bool;   // Impact vibrator fault (CL03)
      motor_client_04_fault : Bool;   // Belt conveyor A fault (CL04)
      motor_client_05_fault : Bool;   // Air knife fault (CL05)
      motor_client_06_fault : Bool;   // Belt conveyor B fault (CL06)
      motor_client_07_fault : Bool;   // Shradder 1 fault (CL07)
      motor_client_08_fault : Bool;   // Shradder vibrator fault (CL08)
      motor_client_09_fault : Bool;   // Belt conveyor C fault (CL09)
      motor_client_10_fault : Bool;   // Rotex screen fault (CL10)
      motor_client_11_fault : Bool;   // free db3_dbx_15_3
      motor_client_12_fault : Bool;   // free db3_dbx_15_3
      motor_client_13_fault : Bool;   // Apron conveyor B fault (CL13)
      motor_client_14_fault : Bool;   // Shradder 2 fault (CL14)
      motor_client_15_fault : Bool;   // Belt conveyor D fault (CL15)
      motor_client_16_fault : Bool;   // Belt conveyor E fault (CL16)
      motor_client_17_fault : Bool;   // fr ee (CL17)
      motor_client_18_fault : Bool;   // [db3.dbx16.2]
      motor_client_19_fault : Bool;   // Primary shradder fault (CL19)
      BWF01_Fault_Control : Bool;   // BWF 01 Control sytem fault
      BWF02_Fault_Control : Bool;   // BWF 02 Control sytem fault
      Emergency_module_fault : Bool;   // Emergency module alarm, reset the module
      "Simulation enabled" : Bool;   // Simulation enabled
      Prealarms_FN01 : Bool;   // Prealarm stop FN-01
      Prealarms_FN04 : Bool;   // Prealarm stop FN-04
      Aux_Inverter_Fault : Bool;   // Auxiliary inverter FAULT
      PLC_DIAGNOSTIC_FAULT : Bool;   // PLC Hardware diagnostic fault FAULT
      EmergencyStopTC1_2 : Bool;
      BC01_Absorbption_OFR : Bool;
      MC04_Absorbption_OFR : Bool;
      Free_011 : Bool;
      Free_012 : Bool;
      Free_013 : Bool;
      Free_014 : Bool;
      Free_015 : Bool;
      Free_016 : Bool;
      Free_017 : Bool;
      Free_018 : Bool;
      Free_019 : Bool;
      BC01_INV : Bool;   // Fault Inverter BC01
      RD01_INV : Bool;   // Fault Inverter RD01
      MC04_INV : Bool;   // Fault Inverter MC04
      VS01_INV : Bool;   // Fault Inverter VS01
      FN02_INV : Bool;   // Fault Inverter FN02
      FN01_INV : Bool;   // Fault Inverter FN01
      FN03_INV : Bool;   // Fault Inverter FN03
      FN04_INV : Bool;   // Fault Inverter FN04
      Aux_INV : Bool;   // Fault Inverter Auxilary
      ER01_run : Bool;   // feedback allarm ER01
      TC04_OFR : Bool;   // TC04 out of range
      TC05_OFR : Bool;   // TC05 out of range
      TC09_OFR : Bool;   // TC09 out of range
      TC10_OFR : Bool;   // TC10 out of range
      Flow_rate_BWF01_OFR : Bool;   // Flow rate BWF01 out of range
      Flow_rate_BWF02_OFR : Bool;   // Flow rate BWF02 out of range
      Level_BWF01_OFR : Bool;   // Level BWF01 out of range
      Level_BWF02_OFR : Bool;   // Level BWF02 out of range
      TC01_OFR : Bool;   // TC01 out of range
      TC02_OFR : Bool;   // TC02 out of range
      TC03_OFR : Bool;   // TC03 out of range
      TC06_OFR : Bool;   // TC06 out of range
      TC07_OFR : Bool;   // TC07 out of range
      ZT01_OFR : Bool;   // ZT01 out of range
      PSH01_OFR : Bool;   // PSH01 out of range
      PSH02_OFR : Bool;   // PSH02 out of range
      PSH03_OFR : Bool;   // PSH03 out of range
      Ro01_OFR : Bool;   // Ro01 out of range
      RO02_OFR : Bool;   // RO02 out of range
      RO03_OFR : Bool;   // RO03 out of range
      RO04_OFR : Bool;   // RO04 out of range
      BR01_Gas_OFR : Bool;   // BR01 Gas
      BR01_Air_OFR : Bool;   // BR01 Air
      Massico_Gas_OFR : Bool;   // Gas out of range
      Massico_Air_OFR : Bool;   // Air out of range
      MV05_OFR : Bool;   // MV05 out of range
      MV06_OFR : Bool;   // MV06 out of range
      MV04A_OFR : Bool;   // MV04A out of range
      MV04B_OFR : Bool;   // MV04B out of range
      FN02_Absorbption_OFR : Bool;   // FN02 Absorbption out of range
      FN04_Absorbption_OFR : Bool;   // FN04 Absorbption out of range
      RD01_Absorbption_OFR : Bool;   // RD01 Absorbption out of range
      FN01_Absorbption_OFR : Bool;   // FN01 Absorbption out of range
      BF01_OFR : Bool;   // BF01 out of range
      PC01_OFR : Bool;   // PC01 out of range
      BF02_OFR : Bool;   // BF02 out of range
      Pot_MV01_OFR : Bool;   // Pot MV01 out of range
      Pot_MV02_OFR : Bool;   // Pot MV02 out of range
      Pot_MV03_OFR : Bool;   // Pot MV03 out of range
      Pot_MV05_OFR : Bool;   // Pot MV05 out of range
      Pot_MV06_OFR : Bool;   // Pot MV06 out of range
   END_VAR
BEGIN
END_DATA_BLOCK

DATA_BLOCK "Coeff"   // DB4
{ S7_Optimized_Access := 'FALSE' }
VERSION : 0.1
   VAR
      ZERO_BWF2_FEEDER_FLOW_RATE : Int := 0;   // (COEFF_A_FR01)
      COEFF_BWF2_FEEDER_FLOW_RATE : Int := 151;   // (COEFF_A_MVT01)
      ZERO_BWF1_HOPPER_LEVEL : Int := 0;   // (COEFF_A_R003)
      COEFF_BWF1_HOPPER_LEVEL : Int := 101;   // (ZERO_A_R003)
      ZERO_BWF2_HOPPER_LEVEL : Int := 0;   // (Min_DP_PC03)
      COEFF_BWF2_HOPPER_LEVEL : Int := 101;   // (O2_Using_Code)
      ZERO_TC01 : Int := 0;   // (ZERO_TC1)
      COEFF_TC01 : Int := 1330;   // (COEFF_TC1)
      ZERO_TC02 : Int := 0;   // (ZERO_TC03)
      COEFF_TC02 : Int := 1330;   // (COEFF_TC03)
      ZERO_TC03 : Int := 0;   // (COEFF_R004)
      COEFF_TC03 : Int := 1330;   // (ZERO_R004)
      ZERO_TC06 : Int := 0;   // (ZERO_TC04)
      COEFF_TC06 : Int := 1100;   // (COEFF_TC04)
      ZERO_TC07 : Int := 0;   // (ZERO_TC05)
      COEFF_TC07 : Int := 1330;   // (COEFF_TC05)
      ZERO_ZT01 : Int := -3900;   // (ZERO_T500000)
      COEFF_ZT01 : Int := 282;   // (COEFF_T500000)
      ZERO_PSH01 : Int := 0;   // (ZERO_POT_BR01)
      COEFF_PSH01 : Int := 100;   // (COEFF_POT_BR01)
      ZERO_PSH02 : Int := 1;   // (COEFF_TC06)
      COEFF_PSH02 : Int := 100;   // (ZER_TC06)
      ZERO_R01 : Int := 0;   // (ZERO_PC_03)
      COEFF_R01 : Int := 250;   // (COEFF_PC_03)
      ZERO_R02 : Int := 0;   // (ZERO_PC01)
      COEFF_R02 : Int := 250;   // (COEFF_PC01)
      ZERO_R03 : Int := 0;   // (ZERO_PC02)
      COEFF_R03 : Int := 250;   // (COEFF_PC02)
      ZERO_R04 : Int := 0;   // (ZERO_RO02)
      COEFF_R04 : Int := 250;   // (COEFF_RO02)
      ZERO_TRASM_GAS_BR01 : Int := 0;   // (ZERO_RO01)
      COEFF_TRASM_GAS_BR01 : Int := 100;   // (COEFF_RO01)
      ZERO_TRASM_AIR_BR01 : Int := 0;   // (ZERO_GASM0000)
      COEFF_TRASM_AIR_BR01 : Int := 100;   // (COEFF_GASM0000)
      ZERO_FLOW_GAS_BR01 : Int := 0;   // (ZERO_POT_MV01)
      COEFF_FLOW_GAS_BR01 : Int := 480;   // (COEFF_POT_MV01)
      ZERO_FLOW_AIR_BR01 : Int := 0;   // (ZERO_POT_MV02)
      COEFF_FLOW_AIR_BR01 : Int := 8000;   // (COEFF_POT_MV02)
      ZERO_TRASM_MV05 : Int := 0;   // (ZERO_POT_MV03)
      COEFF_TRASM_MV05 : Int := 9600;   // (COEFF_POT_MV03)
      ZERO_TRASM_MV02 : Int := 0;   // (ZERO_POT_MV04)
      COEFF_TRASM_MV02 : Int := 290;   // (COEFF_POT_MV04)
      ZERO_TRASM_MV06 : Int := 0;   // (Zero_pot_VG01)
      FREE : Int := 0;   // (Coeff_pot_VG01)
      FREE_1 : Int := -2600;   // (SETPOINT_PC03)
      COEFF_TRASM_MV04 : Int := 120;
      ZERO_FAN_A_FN02 : Int := 0;
      COEFF_FAN_A_FN02 : Int := 178;
      ZERO_ASPIRATOR_A_FN04 : Int := 0;
      COEFF_ASPIRATOR_A_FN04 : Int := 300;
      ZERO_DRUM_A_RD01 : Int := 0;
      COEFF_DRUM_A_RD01 : Int := 81;
      ZERO_FAN_A_FN01 : Int := 0;
      COEFF_FAN_A_FN01 : Int := 240;
      ZERO_TC04 : Int := 0;
      COEFF_TC04 : Int := 250;
      ZERO_TC05 : Int := 0;
      COEFF_TC05 : Int := 250;
      ZERO_DP01 : Int := 0;
      COEFF_DP01 : Int := 250;
      ZERO_DP02 : Int := 0;
      COEFF_DP02 : Int := 500;
      ZERO_PC01 : Int := -14670;
      COEFF_PC01 : Int := 4000;
      ZERO_TC09 : Int := 0;
      COEFF_TC09 : Int := 1330;
      ZERO_MV04B : Int := -2600;
      COEFF_MV04B : Int := 120;
      FREE_W130 : Int := 0;
      DP_01_SOGLIA_1 : Int := 50;
      DP_01_SOGLIA_2 : Int := 0;
      DP_01_SOGLIA_3 : Int := 0;
      DP_01_SOGLIA_4 : Int := 0;
      DP_01_PAUSA_SOGLIA_1 : S5Time := S5T#4S;
      DP_01_PAUSA_SOGLIA_2 : S5Time := S5T#0MS;
      DP_01_PAUSA_SOGLIA_3 : S5Time := S5T#0MS;
      DP_01_PAUSA_SOGLIA_4 : S5Time := S5T#0MS;
      DP_01_PAUSA_SOGLIA_5 : S5Time := S5T#0MS;
      DP_01_LAVORO_SOGLIA_1 : S5Time := S5T#200MS;
      DP_01_LAVORO_SOGLIA_2 : S5Time := S5T#0MS;
      DP_01_LAVORO_SOGLIA_3 : S5Time := S5T#0MS;
      DP_01_LAVORO_SOGLIA_4 : S5Time := S5T#0MS;
      DP_01_LAVORO_SOGLIA_5 : S5Time := S5T#0MS;
      DP_02_SOGLIA_1 : Int := 0;
      DP_02_SOGLIA_2 : Int := 0;
      DP_02_SOGLIA_3 : Int := 0;
      DP_02_SOGLIA_4 : Int := 0;
      DP_02_PAUSA_SOGLIA_1 : S5Time := S5T#0MS;
      DP_02_PAUSA_SOGLIA_2 : S5Time := S5T#0MS;
      DP_02_PAUSA_SOGLIA_3 : S5Time := S5T#0MS;
      DP_02_PAUSA_SOGLIA_4 : S5Time := S5T#0MS;
      DP_02_PAUSA_SOGLIA_5 : S5Time := S5T#0MS;
      DP_02_LAVORO_SOGLIA_1 : S5Time := S5T#0MS;
      DP_02_LAVORO_SOGLIA_2 : S5Time := S5T#0MS;
      DP_02_LAVORO_SOGLIA_3 : S5Time := S5T#0MS;
      DP_02_LAVORO_SOGLIA_4 : S5Time := S5T#0MS;
      DP_02_LAVORO_SOGLIA_5 : S5Time := S5T#0MS;
      FREE_2 : Int := 0;
      FREE_3 : Int := 0;
      SET_PC01 : Int := -35;
      ZERO_TRASM_MV03 : Int := 0;   // (ZERO_POT_MV03)
      COEFF_TRASM_MV03 : Int := 354;   // (COEFF_POT_MV03)
      ZERO_TRASM_MV01 : Int := 0;   // (ZERO_POT_MV03)
      COEFF_TRASM_MV01 : Int := 465;   // (COEFF_POT_MV03)
      ZERO_BWF1_FEEDER_FLOW_RATE : Int := 0;   // (COEFF_A_FR01)
      COEFF_BWF1_FEEDER_FLOW_RATE : Int := 151;   // (COEFF_A_MVT01)
      Selez_Escl_filtri : Int := 3;
      ZERO_TC10 : Int := 0;
      COEFF_TC10 : Int := 0;
      Zero_PSH03 : Int := 0;
      Coeff_PSH03 : Int := -100;
      Zero_MV06 : Int := 0;
      Coeff_MV06 : Int := 900;
      COEFF_free4 : Int := 0;
      COEFF_free5 : Int := 0;
      COEFF_free6 : Int := 0;
      COEFF_free7 : Int := 0;
      COEFF_free8 : Int := 0;
      COEFF_free9 : Int := 0;
      COEFF_free10 : Int := 0;
      COEFF_free11 : Int := 0;
      COEFF_free12 : Int := 0;
      COEFF_free13 : Int := 0;
      COEFF_free14 : Int := 0;
      COEFF_free15 : Int := 0;
      COEFF_free16 : Int := 0;
      COEFF_free17 : Int := 0;
      COEFF_free18 : Int := 0;
      COEFF_free19 : Int := 0;
   END_VAR
BEGIN
END_DATA_BLOCK

DATA_BLOCK "Stechio"   // DB5
{ S7_Optimized_Access := 'FALSE' }
VERSION : 0.1
   VAR
      Set_stechio : Real := 9.5;   // Desired stoichiometer ratio coefficient setpoint
      Real_stechio : Real := 10.91781;   // Reset working hours after recording the data in the DB
      PID_GAIN : Real := -1.6;   // PID proportional part
      PID_TI : Time := T#6S;   // Integration time
      PID_TD : Time := T#8S;   // Derivative time
      Limite_min : Real := -20.0;   // Stoichiometric correction minimum limit
      Limite_MAX : Real := 20.0;   // Stoichiometric correction maximum limit
      Sign_lim_min : Bool := FALSE;   // Ratio flag too low - Air defect
      Sign_lim_MAX : Bool := TRUE;   // Ratio flag too high Excess air
      Consumo_GAS : Real := 3014.389;
      Consumo_GAS_TOTALE : Real := 46.74721;
      Prodotto1_Passato : Real := 2185.2;
      Prodotto2_Passato : Real := 34.0;
      Free46 : Real := 0.0;
      Gas_crv0_4 : Int := 0;
      Gas_crv5_9 : Int := 20;
      Gas_crv10_14 : Int := 31;
      Gas_crv15_19 : Int := 34;
      Gas_crv20_24 : Int := 38;
      Gas_crv25_29 : Int := 43;
      Gas_crv30_34 : Int := 46;
      Gas_crv35_39 : Int := 52;
      Gas_crv40_44 : Int := 100;
      Gas_crv45_49 : Int := 100;
      Gas_crv50_54 : Int := 100;
      Gas_crv55_59 : Int := 100;
      Gas_crv60_64 : Int := 100;
      Gas_crv65_69 : Int := 100;
      Gas_crv70_74 : Int := 100;
      Gas_crv75_79 : Int := 100;
      Gas_crv80_84 : Int := 100;
      Gas_crv85_89 : Int := 100;
      Gas_crv90_94 : Int := 100;
      Gas_crv95_100 : Int := 100;
      Free90 : Int := 0;
      Free92 : Int := 0;
      Free94 : Int := 0;
      Free96 : Int := 0;
      Free98 : Int := 0;
      Portata_Aria_100 : Real := 16#0000_1388;
      Portata_Aria_richiesta : Real := 0.0;
      Errore_Portata_Aria : Real := 0.0;
      Free112 : Real := 0.0;
      Free116 : Real := 0.0;
      Free120 : Real := 0.0;
   END_VAR
BEGIN
END_DATA_BLOCK

DATA_BLOCK "WorkData"   // DB6
{ S7_Optimized_Access := 'FALSE' }
VERSION : 0.1
   VAR
      W0 : Int;
      W1 : Int;
      W2 : Int;
      W3 : Int;
      W4 : Int;
      W5 : Int;
      Burner_PID_Result : Int;
      W7 : Int;
      W8 : Int;
      W9 : Int;
      R1State : Int;
      BR01_State : Int;
      BR01_CleanTime : Int;
      W13 : Int;
      W14 : Int;
      W15 : Int;
      W16 : Int;
      W17 : Int;
      W18 : Int;
      W19 : Int;
      W20 : Int;
      W21 : Int;
      W22 : Int;
      W23 : Int;
      W24 : Int;
      W25 : Int;
      W26 : Int;
      W27 : Int;
      W28 : Int;
      W29 : Int;
      W30 : Int;
      W31 : Int;
      W32 : Int;
      W33 : Int;
      W34 : Int;
      W35 : Int;
      W36 : Int;
      W37 : Int;
      W38 : Int;
      W39 : Int;
      W40 : Int;
      W41 : Int;
      W42 : Int;
      W43 : Int;
      W44 : Int;
      W45 : Int;
      W46 : Int;
      W47 : Int;
      W48 : Int;
      W49 : Int;
   END_VAR
BEGIN
END_DATA_BLOCK

DATA_BLOCK "ENCODER PEW336"   // DB7
{ S7_Optimized_Access := 'FALSE' }
VERSION : 0.0
BEGIN
END_DATA_BLOCK

DATA_BLOCK "Memory encoder"   // DB8
{ S7_Optimized_Access := 'FALSE' }
VERSION : 0.1
   VAR
      Encoder_CH00 : DInt;
      Encoder_CH01 : DInt;
      Encoder_CH02 : DInt;
      Encoder_CH03 : DInt;
      Encoder_CH04 : DInt;
      Encoder_CH05 : DInt;
      Encoder_CH06 : DInt;
      Encoder_CH07 : DInt;
      Test : DInt;
      Encoder_CH00_10 : Int;
      Encoder_CH01_10 : Int;
      Encoder_CH02_10 : Int;
      Encoder_CH03_10 : Int;
      Encoder_CH04_10 : Int;
      Encoder_CH05_10 : Int;
      Encoder_CH06_10 : Int;
      Encoder_CH07_10 : Int;
   END_VAR
BEGIN
END_DATA_BLOCK

DATA_BLOCK "hours motors"   // DB9
{ S7_Optimized_Access := 'FALSE' }
VERSION : 0.1
   VAR
      CLIENT_MOTOR_1_MIN : Int;
      CLIENT_MOTOR_1_HOUR : Int;
      CLIENT_MOTOR_2_MIN : Int;
      CLIENT_MOTOR_2_HOUR : Int;
      CLIENT_MOTOR_3_MIN : Int;
      CLIENT_MOTOR_3_HOUR : Int;
      CLIENT_MOTOR_4_MIN : Int;
      CLIENT_MOTOR_4_HOUR : Int;
      CLIENT_MOTOR_5_MIN : Int;
      CLIENT_MOTOR_5_HOUR : Int;
      CLIENT_MOTOR_6_MIN : Int;
      CLIENT_MOTOR_6_HOUR : Int;
      CLIENT_MOTOR_7_MIN : Int;
      CLIENT_MOTOR_7_HOUR : Int;
      CLIENT_MOTOR_8_MIN : Int;
      CLIENT_MOTOR_8_HOUR : Int;
      CLIENT_MOTOR_9_MIN : Int;
      CLIENT_MOTOR_9_HOUR : Int;
      CLIENT_MOTOR_10_MIN : Int;
      CLIENT_MOTOR_10_HOUR : Int;
      CLIENT_MOTOR_11_MIN : Int;
      CLIENT_MOTOR_11_HOUR : Int;
      CLIENT_MOTOR_12_MIN : Int;
      CLIENT_MOTOR_12_HOUR : Int;
      CLIENT_MOTOR_13_MIN : Int;
      CLIENT_MOTOR_13_HOUR : Int;
      CLIENT_MOTOR_14_MIN : Int;
      CLIENT_MOTOR_14_HOUR : Int;
      CLIENT_MOTOR_15_MIN : Int;
      CLIENT_MOTOR_15_HOUR : Int;
      CLIENT_MOTOR_16_MIN : Int;
      CLIENT_MOTOR_16_HOUR : Int;
      CLIENT_MOTOR_17_MIN : Int;
      CLIENT_MOTOR_17_HOUR : Int;
      CLIENT_MOTOR_18_MIN : Int;
      CLIENT_MOTOR_18_HOUR : Int;
      CLIENT_MOTOR_19_MIN : Int;
      CLIENT_MOTOR_19_HOUR : Int;
      BC_01_MIN : Int;
      BC_01_HOUR : Int;
      RD_01_MIN : Int;
      RD_01_HOUR : Int;
      RD_01_FAN_MIN : Int;
      RD_01_FAN_HOUR : Int;
      MC_03_MIN : Int;
      MC_03_HOUR : Int;
      MC_04_MIN : Int;
      MC_04_HOUR : Int;
      MC_05_MIN : Int;
      MC_05_HOUR : Int;
      VS_01_MIN : Int;
      VS_01_HOUR : Int;
      SC_12_MIN : Int;
      SC_12_HOUR : Int;
      FN_02_MIN : Int;
      FN_02_HOUR : Int;
      VR_01_MIN : Int;
      VR_01_HOUR : Int;
      FN_01_MIN : Int;
      FN_01_HOUR : Int;
      VR_02_MIN : Int;
      VR_02_HOUR : Int;
      CH_01_MIN : Int;
      CH_01_HOUR : Int;
      FN_03_MIN : Int;
      FN_03_HOUR : Int;
      FN_06_MIN : Int;
      FN_06_HOUR : Int;
      SC_01_MIN : Int;
      SC_01_HOUR : Int;
      FN_01_FAN_MIN : Int;
      FN_01_FAN_HOUR : Int;
      LD_01_MIN : Int;
      LD_01_HOUR : Int;
      LD_01_VIB_MIN : Int;
      LD_01_VIB_HOUR : Int;
      SC_10_MIN : Int;
      SC_10_HOUR : Int;
      SC_11_MIN : Int;
      SC_11_HOUR : Int;
      FN_04_MIN : Int;
      FN_04_HOUR : Int;
      VR_03_MIN : Int;
      VR_03_HOUR : Int;
      VR_04_MIN : Int;
      VR_04_HOUR : Int;
      VR_05_MIN : Int;
      VR_05_HOUR : Int;
      VR_06_MIN : Int;
      VR_06_HOUR : Int;
      FN_05_MIN : Int;
      FN_05_HOUR : Int;
      INDEX : Int;
      HOUR : Int;
      MINUTE : Int;
   END_VAR
BEGIN
END_DATA_BLOCK

DATA_BLOCK "Data2"   // DB10
{ S7_Optimized_Access := 'FALSE' }
VERSION : 0.1
   VAR
      Set_TH : Int := 10;
      Set_MAX_TH : Int := 10;
      Free4 : Int := 0;
      Free5 : Int := 0;
      Free8 : Int := 0;
      Free10 : Int := 0;
      Free12 : Int := 0;
      Free14 : Int := 0;
      Free16 : Int := 0;
      Free18 : Int := 0;
      Free20 : Int := 0;
      Free22 : Int := 0;
      Free_111 : Int := 0;
      Free_112 : Int := 0;
      Free_113 : Int := 0;
      Free_114 : Int := 0;
      Free_115 : Int := 0;
      Free_116 : Int := 0;
      Free_117 : Int := 0;
      Free_118 : Int := 0;
      Set_MAX_TH1 : Int := 15;
      Set_MAX_TH2 : Int := 15;
      Set_MAX_TH3 : Int := 0;
      Set_MAX_TH4 : Int := 0;
      Set_MAX_TH5 : Int := 0;
      Set_MAX_TH6 : Int := 0;
      Set_MAX_TH7 : Int := 0;
      Set_MAX_TH8 : Int := 0;
      Set_MAX_TH9 : Int := 0;
      Set_MAX_TH10 : Int := 0;
      Free_1 : Int := 0;
      Free_12 : Int := 0;
      Free_13 : Int := 0;
      Free_14 : Int := 0;
      Free_15 : Int := 0;
      Free_16 : Int := 0;
      Free_17 : Int := 0;
      Free_18 : Int := 0;
      Free_19 : Int := 0;
      Free_110 : Int := 0;
   END_VAR
BEGIN
END_DATA_BLOCK

DATA_BLOCK "Instance for FB12"   // DB12
{ S7_Optimized_Access := 'FALSE' }
VERSION : 0.1
   VAR
      DB_VAR : Int;   // Variabile jolly provvisoria / Jolly temporary tag
   END_VAR
BEGIN
END_DATA_BLOCK

DATA_BLOCK "SIMULATIONDB"   // DB27
{ S7_Optimized_Access := 'TRUE' }
VERSION : 0.1
   VAR
      "TIMER 1" : IEC_TIMER;
      "TIMER 2" : IEC_TIMER;
      "TIMER 3" : IEC_TIMER;
      "TIMER 4" : IEC_TIMER;
      "TIMER 5" : IEC_TIMER;
      "TIMER 6" : IEC_TIMER;
      "TIMER 7" : IEC_TIMER;
      "TIMER 8" : IEC_TIMER;
      "TIMER 9" : IEC_TIMER;
      "TIMER 10" : IEC_TIMER;
   END_VAR
BEGIN
END_DATA_BLOCK

DATA_BLOCK "Manage_TC1_2"   // DB39
{ S7_Optimized_Access := 'FALSE' }
VERSION : 0.1
   VAR
      EnableTC01 : Bool := true;
      EnableTC02 : Bool := true;
      PID_Ref_Temp : Real;
      EmergencyStop : Bool;
   END_VAR
BEGIN
END_DATA_BLOCK

DATA_BLOCK "HMI_DB"   // DB41
{ S7_Optimized_Access := 'FALSE' }
VERSION : 0.1
   VAR
      Counter_StopBurner : Int;   // Counter for Burner Off with cycle On
      Counter_GasConsumption : Int;
      Counter_TotalProduction : Real;
      Counter_PartialProduction : Real;   // Produced Tons
      InternalCounter_StopBurner : Int;
      InternalCounter_TotalProduction : Real;
      InternalCounter_PartialProduction : Real;
      InternalCounter_GasConsumption : Int;
      memoBurnerON : Bool;
      FN01_Preheating_1st_step_temperature : Real;
      FN01_Preheating_2nd_step_temperature : Real;
      FN01_Preheating_3rd_step_temperature : Real;
      FN01_Preheating_4th_step_temperature : Real;
      FN01_Preheating_1st_step_speed : Int;
      FN01_Preheating_2nd_step_speed : Int;
      FN01_Preheating_3rd_step_speed : Int;
      FN01_Preheating_4th_step_speed : Int;
      PreheatingControl_Enabled : Bool;
      ResetCounter_StopBurner : Bool;
      ResetCounter_GasConsumption : Bool;
      ResetCounter_PartialProduction : Bool;
      ResetCounter_TotalProduction : Bool;
      ResetEncoderProcedure_MV01 : Bool;
      ResetEncoderProcedure_MV03 : Bool;
      SET_PERC_BC01 : Int;
      SET_PERC_MC04 : Int;
      Amp_BC01 : Int;
      Amp_MC04 : Int;
   END_VAR
BEGIN
END_DATA_BLOCK

DATA_BLOCK "fill_unit1"   // DB91
{ S7_Optimized_Access := 'FALSE' }
VERSION : 1.0
BEGIN
   MOD_ADR := WORD#16#0150;
   CH_ADR := DWORD#16#0000_0A80;
END_DATA_BLOCK

DATA_BLOCK "Word_inputs"   // DB100
{ S7_Optimized_Access := 'FALSE' }
VERSION : 0.1
   VAR
      word1 : Word;
      word2 : Word;
      word3 : Word;
      word4 : Word;
      word5 : Word;
      word6 : Word;
      word7 : Word;
      word8 : Word;
      word9 : Word;
      word10 : Word;
   END_VAR
BEGIN
END_DATA_BLOCK

DATA_BLOCK "Word_outputs"   // DB101
{ S7_Optimized_Access := 'FALSE' }
VERSION : 0.1
   VAR
      WORD1 : Word;
      WORD2 : Word;
      WORD3 : Word;
      WORD4 : Word;
      WORD5 : Word;
      WORD6 : Word;
      WORD7 : Word;
      WORD8 : Word;
      WORD9 : Word;
      WORD10 : Word;
      WORD11 : Word;
   END_VAR
BEGIN
END_DATA_BLOCK

DATA_BLOCK "DATA_PID"   // DB150
{ S7_Optimized_Access := 'FALSE' }
VERSION : 0.1
   VAR
      TI_FN02 : Time;
      GAIN_FN02 : Real;
   END_VAR
BEGIN
END_DATA_BLOCK

DATA_BLOCK "DB200"   // DB200
{ S7_Optimized_Access := 'FALSE' }
VERSION : 0.1
   VAR
      DB_VAR : Date_And_Time;
      DB_VAR1 : Date_And_Time;
      test : Date;
      test1 : Time_Of_Day;
      test2 : Date := D#2011-12-06;
   END_VAR
BEGIN
END_DATA_BLOCK

// folder: FOR HMI

DATA_BLOCK "Motors"   // DB11
{ S7_Optimized_Access := 'FALSE' }
VERSION : 0.1
   VAR
      BC01 : "Motor";
      RD01 : "Motor";
      RD01_FAN : "Motor";
      SPARE : "Motor";
      MC04 : "Motor";
      MC05 : "Motor";
      VS01 : "Motor";
      SC12 : "Motor";
      AUX_INV : "Motor";
      MV01 : "Motorized Valve";
      MV02 : "Motorized Valve";
      MV03 : "Motorized Valve";
      MV04 : "Motorized Valve";
      MV05 : "Motorized Valve";
      MV06 : "Motorized Valve";
      FN02 : "Motor";
      VR01 : "Motor";
      FN01 : "Motor";
      VR02 : "Motor";
      CH01 : "Motor";
      FN03 : "Motor";
      FN06 : "Motor";
      SC1 : "Motor";
      FN01_FAN : "Motor";
      LD01_MF : "Motor";
      LD01_VB : "Motor";
      SC10 : "Motor";
      SC11 : "Motor";
      FN04 : "Motor";
      VR03 : "Motor";
      VR04 : "Motor";
      VR05 : "Motor";
      VR06 : "Motor";
      FN05 : "Motor";
      ER01 : "Motor";
      BWF01 : "Client Motor";
      BWF02 : "Client Motor";
      PV_14 : "Valve";
      PV_01 : "PV_2_GATE";
      PV_02 : "PV_2_GATE";
      PV_03 : "PV_1_GATE";
      PV_04 : "PV_1_GATE";
      BR_01 : "BR-01";
      EV_03 : "Valve";
   END_VAR
BEGIN
END_DATA_BLOCK

